(* Logix 5000 project; controller Drives_Line1 1756-L72 rev 20.13; software revision 20.04 *)

TASK Medium (periodic, rate 50 ms, priority 10, watchdog 1000 ms) : P00_Line, P01_Entry_Zone, P02_Exit_Zone, P10_Unwinder_1, P11_Unwinder_2, P12_Pinchroll_1, P13_Pinchroll_2, P14_Bridle_01

MODULES
   Local : 1756-L72 (ICP 0, rev 20.13)
      Master_Line_1 : 1756-L72 (ICP 5, rev 20.1, $099675bf$ RPI 20 ms, $797531a6$ RPI 20 ms, $6b587a51$ RPI 20 ms)
      EN2TR : vendor 1 type 12 code 200 (ICP 1, Ethernet 192.168.1.6, rev 3.1, Input RPI 500 ms)
         Drive_Bridle_04a : vendor 1 type 142 code 2192 (Ethernet 192.168.1.23, rev 7.1, Output RPI 20 ms)
             : vendor 1 type 142 code 8352 (RhinoBP 6, rev 1.6)
             : vendor 1 type 142 code 416 (RhinoBP 7, rev 1.8)
             : vendor 1 type 142 code 16544 (RhinoBP 5, rev 1.1)
             : vendor 1 type 142 code 24736 (RhinoBP 8, rev 1.1)
             : vendor 1 type 142 code 32928 (RhinoBP 13, rev 1.1)
             : vendor 1 type 142 code 33184 (RhinoBP 14, rev 2.5)
             : vendor 1 type 142 code 57760 (RhinoBP 4, rev 1.1)
         Drive_Pinchroll_2 : vendor 1 type 142 code 2192 (Ethernet 192.168.1.13, rev 7.1, Output RPI 20 ms)
             : vendor 1 type 142 code 416 (RhinoBP 7, rev 1.8)
             : vendor 1 type 142 code 57760 (RhinoBP 4, rev 1.1)
             : vendor 1 type 142 code 767 (RhinoBP 1, rev 2.2)
             : vendor 1 type 142 code 32928 (RhinoBP 13, rev 1.1)
             : vendor 1 type 142 code 24736 (RhinoBP 8, rev 1.1)
             : vendor 1 type 142 code 33184 (RhinoBP 14, rev 2.5)
             : vendor 1 type 142 code 8352 (RhinoBP 6, rev 1.6)
             : vendor 1 type 142 code 16544 (RhinoBP 5, rev 1.1)
         Drive_Pinchroll_3 : vendor 1 type 142 code 2192 (Ethernet 192.168.1.26, rev 5.1, Output RPI 20 ms)
             : vendor 1 type 142 code 33184 (RhinoBP 14, rev 2.4)
             : vendor 1 type 142 code 24736 (RhinoBP 8, rev 1.1)
             : vendor 1 type 142 code 16544 (RhinoBP 5, rev 1.1)
             : vendor 1 type 142 code 32928 (RhinoBP 13, rev 1.1)
             : vendor 1 type 142 code 8352 (RhinoBP 6, rev 1.6)
             : vendor 1 type 142 code 57760 (RhinoBP 4, rev 1.1)
             : vendor 1 type 142 code 416 (RhinoBP 7, rev 1.8)
         Drive_Bridle_02a : vendor 1 type 142 code 2192 (Ethernet 192.168.1.18, rev 7.1, Output RPI 20 ms)
             : vendor 1 type 142 code 416 (RhinoBP 7, rev 1.8)
             : vendor 1 type 142 code 16544 (RhinoBP 5, rev 1.1)
             : vendor 1 type 142 code 24736 (RhinoBP 8, rev 1.1)
             : vendor 1 type 142 code 33184 (RhinoBP 14, rev 2.5)
             : vendor 1 type 142 code 8352 (RhinoBP 6, rev 1.6)
             : vendor 1 type 142 code 32928 (RhinoBP 13, rev 1.1)
             : vendor 1 type 142 code 57760 (RhinoBP 4, rev 1.1)
         Drive_Unwinder_1 : vendor 1 type 142 code 2192 (Ethernet 192.168.1.10, rev 7.1, Output RPI 20 ms)
             : vendor 1 type 142 code 8352 (RhinoBP 6, rev 1.6)
             : vendor 1 type 142 code 33184 (RhinoBP 14, rev 2.5)
             : vendor 1 type 142 code 57760 (RhinoBP 4, rev 1.1)
             : vendor 1 type 142 code 32928 (RhinoBP 13, rev 1.1)
             : vendor 1 type 142 code 767 (RhinoBP 1, rev 2.2)
             : vendor 1 type 142 code 24736 (RhinoBP 8, rev 1.1)
             : vendor 1 type 142 code 416 (RhinoBP 7, rev 1.8)
             : vendor 1 type 142 code 16544 (RhinoBP 5, rev 1.1)
         Drive_Bridle_01a : vendor 1 type 142 code 2192 (Ethernet 192.168.1.14, rev 7.1, Output RPI 20 ms)
             : vendor 1 type 142 code 57760 (RhinoBP 4, rev 1.1)
             : vendor 1 type 142 code 16544 (RhinoBP 5, rev 1.1)
             : vendor 1 type 142 code 8352 (RhinoBP 6, rev 1.6)
             : vendor 1 type 142 code 33184 (RhinoBP 14, rev 2.5)
             : vendor 1 type 142 code 416 (RhinoBP 7, rev 1.8)
             : vendor 1 type 142 code 24736 (RhinoBP 8, rev 1.1)
             : vendor 1 type 142 code 32928 (RhinoBP 13, rev 1.1)
         Drive_Bridle_02b : vendor 1 type 142 code 2192 (Ethernet 192.168.1.19, rev 7.1, Output RPI 20 ms)
             : vendor 1 type 142 code 33184 (RhinoBP 14, rev 2.5)
             : vendor 1 type 142 code 24736 (RhinoBP 8, rev 1.1)
             : vendor 1 type 142 code 416 (RhinoBP 7, rev 1.8)
             : vendor 1 type 142 code 57760 (RhinoBP 4, rev 1.1)
             : vendor 1 type 142 code 16544 (RhinoBP 5, rev 1.1)
             : vendor 1 type 142 code 8352 (RhinoBP 6, rev 1.6)
             : vendor 1 type 142 code 32928 (RhinoBP 13, rev 1.1)
         Drive_Bridle_03a : vendor 1 type 142 code 2192 (Ethernet 192.168.1.20, rev 7.1, Output RPI 20 ms)
             : vendor 1 type 142 code 57760 (RhinoBP 4, rev 1.1)
             : vendor 1 type 142 code 8352 (RhinoBP 6, rev 1.6)
             : vendor 1 type 142 code 33184 (RhinoBP 14, rev 2.5)
             : vendor 1 type 142 code 32928 (RhinoBP 13, rev 1.1)
             : vendor 1 type 142 code 416 (RhinoBP 7, rev 1.8)
             : vendor 1 type 142 code 16544 (RhinoBP 5, rev 1.1)
             : vendor 1 type 142 code 24736 (RhinoBP 8, rev 1.1)
         Drive_Bridle_01c : vendor 1 type 142 code 2192 (Ethernet 192.168.1.16, rev 7.1, Output RPI 20 ms)
             : vendor 1 type 142 code 416 (RhinoBP 7, rev 1.8)
             : vendor 1 type 142 code 8352 (RhinoBP 6, rev 1.6)
             : vendor 1 type 142 code 32928 (RhinoBP 13, rev 1.1)
             : vendor 1 type 142 code 16544 (RhinoBP 5, rev 1.1)
             : vendor 1 type 142 code 24736 (RhinoBP 8, rev 1.1)
             : vendor 1 type 142 code 57760 (RhinoBP 4, rev 1.1)
             : vendor 1 type 142 code 33184 (RhinoBP 14, rev 2.5)
         Drive_Unwinder_2 : vendor 1 type 142 code 2192 (Ethernet 192.168.1.11, rev 7.1, Output RPI 20 ms)
             : vendor 1 type 142 code 416 (RhinoBP 7, rev 1.8)
             : vendor 1 type 142 code 24736 (RhinoBP 8, rev 1.1)
             : vendor 1 type 142 code 767 (RhinoBP 1, rev 2.2)
             : vendor 1 type 142 code 33184 (RhinoBP 14, rev 2.5)
             : vendor 1 type 142 code 57760 (RhinoBP 4, rev 1.1)
             : vendor 1 type 142 code 16544 (RhinoBP 5, rev 1.1)
             : vendor 1 type 142 code 8352 (RhinoBP 6, rev 1.6)
             : vendor 1 type 142 code 32928 (RhinoBP 13, rev 1.1)
         Drive_Bridle_01b : vendor 1 type 142 code 2192 (Ethernet 192.168.1.15, rev 7.1, Output RPI 20 ms)
             : vendor 1 type 142 code 57760 (RhinoBP 4, rev 1.1)
             : vendor 1 type 142 code 416 (RhinoBP 7, rev 1.8)
             : vendor 1 type 142 code 33184 (RhinoBP 14, rev 2.5)
             : vendor 1 type 142 code 8352 (RhinoBP 6, rev 1.6)
             : vendor 1 type 142 code 32928 (RhinoBP 13, rev 1.1)
             : vendor 1 type 142 code 16544 (RhinoBP 5, rev 1.1)
             : vendor 1 type 142 code 24736 (RhinoBP 8, rev 1.1)
         Drive_Pinchroll_1 : vendor 1 type 142 code 2192 (Ethernet 192.168.1.12, rev 7.1, Output RPI 20 ms)
             : vendor 1 type 142 code 57760 (RhinoBP 4, rev 1.1)
             : vendor 1 type 142 code 24736 (RhinoBP 8, rev 1.1)
             : vendor 1 type 142 code 16544 (RhinoBP 5, rev 1.1)
             : vendor 1 type 142 code 8352 (RhinoBP 6, rev 1.6)
             : vendor 1 type 142 code 33184 (RhinoBP 14, rev 2.5)
             : vendor 1 type 142 code 32928 (RhinoBP 13, rev 1.1)
             : vendor 1 type 142 code 416 (RhinoBP 7, rev 1.8)
         Drive_Bridle_03b : vendor 1 type 142 code 2192 (Ethernet 192.168.1.21, rev 7.1, Output RPI 20 ms)
             : vendor 1 type 142 code 32928 (RhinoBP 13, rev 1.1)
             : vendor 1 type 142 code 416 (RhinoBP 7, rev 1.8)
             : vendor 1 type 142 code 16544 (RhinoBP 5, rev 1.1)
             : vendor 1 type 142 code 57760 (RhinoBP 4, rev 1.1)
             : vendor 1 type 142 code 33184 (RhinoBP 14, rev 2.5)
             : vendor 1 type 142 code 8352 (RhinoBP 6, rev 1.6)
             : vendor 1 type 142 code 24736 (RhinoBP 8, rev 1.1)
         Drive_Winder : vendor 1 type 142 code 2192 (Ethernet 192.168.1.27, rev 7.1, Output RPI 20 ms)
             : vendor 1 type 142 code 24736 (RhinoBP 8, rev 1.1)
             : vendor 1 type 142 code 32928 (RhinoBP 13, rev 1.1)
             : vendor 1 type 142 code 416 (RhinoBP 7, rev 1.8)
             : vendor 1 type 142 code 8352 (RhinoBP 6, rev 1.6)
             : vendor 1 type 142 code 57760 (RhinoBP 4, rev 1.1)
             : vendor 1 type 142 code 33184 (RhinoBP 14, rev 2.5)
             : vendor 1 type 142 code 16544 (RhinoBP 5, rev 1.1)
         Drive_Bridle_04c : vendor 1 type 142 code 2192 (Ethernet 192.168.1.25, rev 7.1, Output RPI 20 ms)
             : vendor 1 type 142 code 57760 (RhinoBP 4, rev 1.1)
             : vendor 1 type 142 code 16544 (RhinoBP 5, rev 1.1)
             : vendor 1 type 142 code 33184 (RhinoBP 14, rev 2.5)
             : vendor 1 type 142 code 24736 (RhinoBP 8, rev 1.1)
             : vendor 1 type 142 code 416 (RhinoBP 7, rev 1.8)
             : vendor 1 type 142 code 8352 (RhinoBP 6, rev 1.6)
             : vendor 1 type 142 code 767 (RhinoBP 1, rev 2.2)
             : vendor 1 type 142 code 32928 (RhinoBP 13, rev 1.1)
         Drive_Entry_Accu : vendor 1 type 142 code 2192 (Ethernet 192.168.1.17, rev 9.1, Output RPI 20 ms)
             : vendor 1 type 142 code 57760 (RhinoBP 4, rev 1.1)
             : vendor 1 type 142 code 33184 (RhinoBP 14, rev 2.5)
             : vendor 1 type 142 code 24736 (RhinoBP 8, rev 1.1)
             : vendor 1 type 142 code 8352 (RhinoBP 6, rev 1.6)
             : vendor 1 type 142 code 16544 (RhinoBP 5, rev 1.1)
             : vendor 1 type 142 code 767 (RhinoBP 1, rev 2.2)
             : vendor 1 type 142 code 416 (RhinoBP 7, rev 1.8)
             : vendor 1 type 142 code 32928 (RhinoBP 13, rev 1.1)
         Drive_Exit_Accu : vendor 1 type 142 code 2192 (Ethernet 192.168.1.22, rev 7.1, Output RPI 20 ms)
             : vendor 1 type 142 code 33184 (RhinoBP 14, rev 2.5)
             : vendor 1 type 142 code 8352 (RhinoBP 6, rev 1.6)
             : vendor 1 type 142 code 416 (RhinoBP 7, rev 1.8)
             : vendor 1 type 142 code 24736 (RhinoBP 8, rev 1.1)
             : vendor 1 type 142 code 57760 (RhinoBP 4, rev 1.1)
             : vendor 1 type 142 code 16544 (RhinoBP 5, rev 1.1)
             : vendor 1 type 142 code 32928 (RhinoBP 13, rev 1.1)
         Drive_Bridle_04b : vendor 1 type 142 code 2192 (Ethernet 192.168.1.24, rev 7.1, Output RPI 20 ms)
             : vendor 1 type 142 code 416 (RhinoBP 7, rev 1.8)
             : vendor 1 type 142 code 16544 (RhinoBP 5, rev 1.1)
             : vendor 1 type 142 code 8352 (RhinoBP 6, rev 1.6)
             : vendor 1 type 142 code 57760 (RhinoBP 4, rev 1.1)
             : vendor 1 type 142 code 32928 (RhinoBP 13, rev 1.1)
             : vendor 1 type 142 code 33184 (RhinoBP 14, rev 2.5)
             : vendor 1 type 142 code 24736 (RhinoBP 8, rev 1.1)
         Drive_cu : PowerFlex 755-EENET (Ethernet 192.168.1.28, rev 9.1, Output RPI 20 ms)
             : vendor 1 type 143 code 767 (RhinoBP 1, rev 2.3)
             : vendor 1 type 143 code 9472 (RhinoBP 2, rev 1.4)
             : vendor 1 type 143 code 8352 (RhinoBP 6, rev 1.6)
             : vendor 1 type 143 code 32928 (RhinoBP 13, rev 1.1)
             : vendor 1 type 143 code 33184 (RhinoBP 14, rev 2.5)
             : vendor 1 type 143 code 416 (RhinoBP 4, rev 1.8)
             : vendor 1 type 143 code 16544 (RhinoBP 5, rev 1.1)
END_MODULES

TYPE UDT_Bridle_2M :
STRUCT
   PF755_shaft_a : UDT_PF755;
   PF755_shaft_b : UDT_PF755;
   Cmd : UDT_Commands_Bridle;
   Stat : UDT_Status_Bridle;
   Ctrl : UDT_Control_Bridle_2M;
   Fbdk_shaft_a : UDT_Feedbacks_Bridle;
   Fbdk_shaft_b : UDT_Feedbacks_Bridle;
   Config_shaft_a : UDT_Config_Bridle;
   Config_shaft_b : UDT_Config_Bridle;
   SpdTrim_MPS : REAL;
   SpdTrim_Pct : REAL;
END_STRUCT
END_TYPE

TYPE UDT_Bridle_3M :
STRUCT
   PF755_shaft_a : UDT_PF755;
   PF755_shaft_b : UDT_PF755;
   PF755_shaft_c : UDT_PF755;
   Stat : UDT_Status_Bridle;
   Fbdk_shaft_a : UDT_Feedbacks_Bridle;
   Fbdk_shaft_b : UDT_Feedbacks_Bridle;
   Fbdk_shaft_c : UDT_Feedbacks_Bridle;
   Config_shaft_a : UDT_Config_Bridle;
   Config_shaft_b : UDT_Config_Bridle;
   Config_shaft_c : UDT_Config_Bridle;
END_STRUCT
END_TYPE

TYPE UDT_Commands :
STRUCT
   Line : UDT_Commands_Line;
   Entry : UDT_Commands_Zone;
   Exit : UDT_Commands_Zone;
   Unwinder_1 : UDT_Commands_Unwinder;
   Unwinder_2 : UDT_Commands_Unwinder;
   Pinchroll_1 : UDT_Commands_Pinch;
   Pinchroll_2 : UDT_Commands_Pinch;
   Entry_Accu : UDT_Commands_Accu;
   Bridle_02 : UDT_Commands_Bridle;
   Bridle_03 : UDT_Commands_Bridle;
   Exit_Accu : UDT_Commands_Accu;
   PinchRoll_3 : UDT_Commands_Pinch;
   Winder : UDT_Commands_Winder;
   cu : UDT_Commands_Pinch;
END_STRUCT
END_TYPE

TYPE UDT_Commands_Accu :
STRUCT
   Run : BOOL;
   JogFwd : BOOL;
   JogRev : BOOL;
END_STRUCT
END_TYPE

TYPE UDT_Commands_Bridle :
STRUCT
   Run : BOOL;
   JogFwd : BOOL;
   JogRev : BOOL;
END_STRUCT
END_TYPE

TYPE UDT_Commands_Line :
STRUCT
   Run : BOOL;
   JogFwd : BOOL;
   JogRev : BOOL;
   ResetDrv : BOOL;
   WD_FromMaster : BOOL;
   ApplyFastStop : BOOL;
END_STRUCT
END_TYPE

TYPE UDT_Commands_Pinch :
STRUCT
   Run : BOOL;
   Coupled_shaft_1 : BOOL;
   Coupled_shaft_2 : BOOL;
   JogFwd : BOOL;
   JogRev : BOOL;
   MtrCb : BOOL;
END_STRUCT
END_TYPE

TYPE UDT_Commands_Unwinder :
STRUCT
   RunFwd : BOOL;
   RunRev : BOOL;
   JogFwd : BOOL;
   JogRev : BOOL;
   SetNewDiameter : BOOL;
   HeadToStitch : BOOL;
   HeadToShear : BOOL;
   ResetCoilLength : BOOL;
END_STRUCT
END_TYPE

TYPE UDT_Commands_Winder :
STRUCT
   RunFwd : BOOL;
   RunRev : BOOL;
   JogFwd : BOOL;
   JogRev : BOOL;
   SetNewDiameter : BOOL;
   ResetCoilLength : BOOL;
END_STRUCT
END_TYPE

TYPE UDT_Commands_Zone :
STRUCT
   Run : BOOL;
   JogFwd : BOOL;
   JogRev : BOOL;
   EndToShear : BOOL;
   EndToStitch : BOOL;
   HeadToStitch : BOOL;
   EndToCoiler : BOOL;
   NewStitch : BOOL;
END_STRUCT
END_TYPE

TYPE UDT_Config :
STRUCT
   Unwinder_1 : UDT_Config_Unwinder;
   Unwinder_2 : UDT_Config_Unwinder;
   Pinchroll_1 : UDT_Config_Pinch;
   Pinchroll_2 : UDT_Config_Pinch;
   Entry_Accu : UDT_Config_Accu;
   Bridle_01a : UDT_Config_Bridle;
   Bridle_01b : UDT_Config_Bridle;
   Bridle_01c : UDT_Config_Bridle;
   Bridle_02a : UDT_Config_Bridle;
   Bridle_02b : UDT_Config_Bridle;
   Bridle_03a : UDT_Config_Bridle;
   Bridle_03b : UDT_Config_Bridle;
   Bridle_04a : UDT_Config_Bridle;
   Bridle_04b : UDT_Config_Bridle;
   Bridle_04c : UDT_Config_Bridle;
   Exit_Accu : UDT_Config_Accu;
   PinchRoll_3 : UDT_Config_Pinch;
   Winder : UDT_Config_Winder;
   Entry : UDT_Config_Zone;
   Exit : UDT_Config_Zone;
   Line : UDT_Config_Line;
END_STRUCT
END_TYPE

TYPE UDT_Config_Accu :
STRUCT
   zGearRatio : REAL;
   zMaxPos : REAL;
   zMinPos : REAL;
   zSyncPos : REAL;
   zJogRef : REAL;
   zAccJog : REAL;
   zDecJog : REAL;
   zJerkJog : REAL;
END_STRUCT
END_TYPE

TYPE UDT_Config_Bridle :
STRUCT
   zGearRatio : REAL;
   DiameterRoll : REAL;
END_STRUCT
END_TYPE

TYPE UDT_Config_Line :
STRUCT
   zAccRate : REAL;
   zDecRate : REAL;
   zJerk : REAL;
   zJogSpd : REAL;
   zJogAccRate : REAL;
   zJogDecRate : REAL;
   zMaxAccDec : REAL;
   zSpdMax : REAL;
END_STRUCT
END_TYPE

TYPE UDT_Config_Pinch :
STRUCT
   zGearRatio : REAL;
   DiameterRoll : REAL;
   zMaxAcc : REAL;
   zMaxDec : REAL;
   zJogRef : REAL;
   zAccJog : REAL;
   zDecJog : REAL;
   zJerkJog : REAL;
END_STRUCT
END_TYPE

TYPE UDT_Config_TM :
STRUCT
   zMinTen : REAL;
   zMaxTen : REAL;
END_STRUCT
END_TYPE

TYPE UDT_Config_Unwinder :
STRUCT
   zGearRatio : REAL;
   zMinDiameter : REAL;
   zMaxDiameter : REAL;
   zMinTension : REAL;
   zMaxTension : REAL;
   zJogRef : REAL;
   zDiamCalcEnblThresh_MPS : REAL;
   zDiamCalcUpdate_Rev : REAL;
   zMotorPwr : REAL;
   zMtrBaseSpd : REAL;
   zAccJog : REAL;
   zDecJog : REAL;
   zJerkJog : REAL;
END_STRUCT
END_TYPE

TYPE UDT_Config_Winder :
STRUCT
   zGearRatio : REAL;
   zMinDiameter : REAL;
   zMaxDiameter : REAL;
   zMinTension : REAL;
   zMaxTension : REAL;
   zJogRef : REAL;
   zDiamCalcEnblThresh_MPS : REAL;
   zDiamCalcUpdate_Rev : REAL;
   zMotorPwr : REAL;
   zMtrBaseSpd : REAL;
   zAccJog : REAL;
   zDecJog : REAL;
   zJerkJog : REAL;
END_STRUCT
END_TYPE

TYPE UDT_Config_Zone :
STRUCT
   zJogRef : REAL;
   zAccJog : REAL;
   zDecJog : REAL;
   zJerkJog : REAL;
   zAccRun : REAL;
   zDecRun : REAL;
   zJerkRun : REAL;
   zMaxAccDec : REAL;
   zMaxSpd : REAL;
END_STRUCT
END_TYPE

TYPE UDT_Control_Accu :
STRUCT
   Run : BOOL;
   JogFwd : BOOL;
   JogRev : BOOL;
   RmpdRefEnable : BOOL;
   URmpdRefEnable : BOOL;
   StartRamp : BOOL;
   TenRegOn : BOOL;
   PosRegOn : BOOL;
   SetSyncPos : BOOL;
   PosRegOutSpd : REAL;
   SpdTrim : REAL;
   FB_CountsPerMM : DINT;
END_STRUCT
END_TYPE

TYPE UDT_Control_Bridle_2M :
STRUCT
   JogFwd : BOOL;
   JogRev : BOOL;
   StartRamp : BOOL;
   RmpdRefEnable : BOOL;
   URmpdRefEnable : BOOL;
   zJogSpd : REAL;
   zJogAccRate : REAL;
   zJogDecRate : REAL;
   zJogJerkRate : REAL;
   zMaxAccDec : REAL;
END_STRUCT
END_TYPE

TYPE UDT_Control_Line :
STRUCT
   Run : BOOL;
   JogFwd : BOOL;
   JogRev : BOOL;
   StartRamp : BOOL;
   RmpdRefEnable : BOOL;
   URmpdRefEnable : BOOL;
   ApplyFastStop : BOOL;
   TenRegOn : BOOL;
   SpdRefRmp : REAL;
END_STRUCT
END_TYPE

TYPE UDT_Control_Pinch :
STRUCT
   Run : BOOL;
   Coupled_shaft_1 : BOOL;
   Coupled_shaft_2 : BOOL;
   JogFwd : BOOL;
   JogRev : BOOL;
   RmpdRefEnable : BOOL;
   URmpdRefEnable : BOOL;
   StartRamp : BOOL;
END_STRUCT
END_TYPE

TYPE UDT_Control_Unwind :
STRUCT
   JogFwd : BOOL;
   JogRev : BOOL;
   RunFwd : BOOL;
   RunRev : BOOL;
   TenRefStallEnbl : BOOL;
   TrimOn : BOOL;
   TrimPos : BOOL;
   TrimNeg : BOOL;
   TenRefOn : BOOL;
   DiamCalcIncEnbl : BOOL;
   DiamCalcDecEnbl : BOOL;
   TensionRef : REAL;
   RunSpdRef : REAL;
   RunSpdRefRate : REAL;
   RunSpdTrim : REAL;
   StartRamp : BOOL;
   RmpdRefEnable : BOOL;
   URmpdRefEnable : BOOL;
   BR : BOOL;
   Fan : BOOL;
END_STRUCT
END_TYPE

TYPE UDT_Control_Winder :
STRUCT
   JogFwd : BOOL;
   JogRev : BOOL;
   RunFwd : BOOL;
   RunRev : BOOL;
   TenRefStallEnbl : BOOL;
   TrimPos : BOOL;
   TrimNeg : BOOL;
   TrimOn : BOOL;
   TenRefOn : BOOL;
   DiamCalcIncEnbl : BOOL;
   DiamCalcDecEnbl : BOOL;
   TensionRef : REAL;
   RunSpdRef : REAL;
   RunSpdRefRate : REAL;
   RunSpdTrim : REAL;
   StartRamp : BOOL;
   RmpdRefEnable : BOOL;
   URmpdRefEnable : BOOL;
   BR : BOOL;
   Fan : BOOL;
END_STRUCT
END_TYPE

TYPE UDT_Control_Zone :
STRUCT
   Run : BOOL;
   JogFwd : BOOL;
   JogRev : BOOL;
   EndToShear : BOOL;
   EndToStitch : BOOL;
   EndToCoiler : BOOL;
   HeadToStitch : BOOL;
   StartRamp : BOOL;
   RmpdRefEnable : BOOL;
   URmpdRefEnable : BOOL;
   ApplyFastStop : BOOL;
   EOC_PosRedef : DINT;
   HOC_PosRedef : DINT;
   SpdRefRmp : REAL;
END_STRUCT
END_TYPE

TYPE UDT_Datalinks_in :
STRUCT
   OutputFrequency : REAL;
   OutputCurrent : REAL;
   OutputVoltage : REAL;
   OutputPower : REAL;
   SRegOutput : REAL;
   PTP_Feedback : DINT;
   LimitedTrqRef : REAL;
   FaultStatusA : DINT;
   FaultStatusB : DINT;
   StartInhibits : DINT;
   P7_Ptc_Sts : DINT;
   P7_DigitalOutSts : DINT;
   P7_DigitalInSts : DINT;
   HomingStatus : DINT;
END_STRUCT
END_TYPE

TYPE UDT_Datalinks_Out :
STRUCT
   TorqueStep : REAL;
   TorqueSp : REAL;
   RegulatorMode : DINT;
   SpeedRegBW : REAL;
   HomingControl : DINT;
   UserHomePos : DINT;
   PID_Setpoint : REAL;
   SpdRegNegLim : REAL;
   SpdRegPosLim : REAL;
   PID_Ctrl : DINT;
   P7_DigOutSetpoint : DINT;
END_STRUCT
END_TYPE

TYPE UDT_Drive_Commands :
STRUCT
   LogicCommand : DINT;
   Stop : BOOL;
   Start : BOOL;
   Jog1 : BOOL;
   ClearFaults : BOOL;
   Forward : BOOL;
   Reverse : BOOL;
   Manual : BOOL;
   AccelTime1 : BOOL;
   AccelTime2 : BOOL;
   DecelTime1 : BOOL;
   DecelTime2 : BOOL;
   SpdRefSel0 : BOOL;
   SpdRefSel1 : BOOL;
   SpdRefSel2 : BOOL;
   CoastStop : BOOL;
   CLimitStop : BOOL;
   Run : BOOL;
   Jog2 : BOOL;
   Reference : REAL;
END_STRUCT
END_TYPE

TYPE UDT_Drive_Status :
STRUCT
   Drive_status : DINT;
   Ready : BOOL;
   Active : BOOL;
   CommandDir : BOOL;
   ActualDir : BOOL;
   Accelerating : BOOL;
   Decelerating : BOOL;
   Alarm : BOOL;
   Faulted : BOOL;
   AtSpeed : BOOL;
   Manual : BOOL;
   SpdRefBit0 : BOOL;
   SpdRefBit1 : BOOL;
   SpdRefBit2 : BOOL;
   SpdRefBit3 : BOOL;
   SpdRefBit4 : BOOL;
   Running : BOOL;
   Jogging : BOOL;
   Stopping : BOOL;
   DCBraking : BOOL;
   DBActive : BOOL;
   SpeedMode : BOOL;
   PositionMode : BOOL;
   TorqueMode : BOOL;
   AtZeroSpeed : BOOL;
   AtHome : BOOL;
   AtLimit : BOOL;
   CurrLimit : BOOL;
   BusFrqReg : BOOL;
   EnableOn : BOOL;
   MotorOL : BOOL;
   Regen : BOOL;
   Feedback : REAL;
END_STRUCT
END_TYPE

TYPE UDT_Entry_Accu :
STRUCT
   PF755 : UDT_PF755;
   Cmd : UDT_Commands_Accu;
   Stat : UDT_Status_Accu;
   Fdbk : UDT_Feedbacks_Accu;
   Sp : UDT_Setpoints_Accu;
   Config : UDT_Config_Accu;
   Ctrl : UDT_Control_Accu;
END_STRUCT
END_TYPE

TYPE UDT_Exit_Accu :
STRUCT
   PF755 : UDT_PF755;
   Cmd : UDT_Commands_Accu;
   Stat : UDT_Status_Accu;
   Fdbk : UDT_Feedbacks_Accu;
   Sp : UDT_Setpoints_Accu;
   Config : UDT_Config_Accu;
   Ctrl : UDT_Control_Accu;
END_STRUCT
END_TYPE

TYPE UDT_Fdbks :
STRUCT
   Unwinder_1 : UDT_Feedbacks_Unwinder;
   Unwinder_2 : UDT_Feedbacks_Unwinder;
   Pinchroll_1 : UDT_Feedbacks_Pinch;
   Pinchroll_2 : UDT_Feedbacks_Pinch;
   Entry_Accu : UDT_Feedbacks_Accu;
   Bridle_01a : UDT_Feedbacks_Bridle;
   Bridle_01b : UDT_Feedbacks_Bridle;
   Bridle_01c : UDT_Feedbacks_Bridle;
   Bridle_02a : UDT_Feedbacks_Bridle;
   Bridle_02b : UDT_Feedbacks_Bridle;
   Bridle_03a : UDT_Feedbacks_Bridle;
   Bridle_03b : UDT_Feedbacks_Bridle;
   Bridle_04a : UDT_Feedbacks_Bridle;
   Bridle_04b : UDT_Feedbacks_Bridle;
   Bridle_04c : UDT_Feedbacks_Bridle;
   Exit_Accu : UDT_Feedbacks_Accu;
   Pinchroll_3 : UDT_Feedbacks_Pinch;
   Winder : UDT_Feedbacks_Winder;
   Line : UDT_Feedbacks_Line;
   Entry : UDT_Feedbacks_Zone;
   Exit : UDT_Feedbacks_Zone;
   cu : UDT_Feedbacks_Pinch;
END_STRUCT
END_TYPE

TYPE UDT_Feedbacks_Accu :
STRUCT
   PvSpeed : REAL;
   PvActualPos : REAL;
   PvActualPosPct : REAL;
   PvSpdRef_MPS : REAL;
   PvSpdRef_RPM : REAL;
END_STRUCT
END_TYPE

TYPE UDT_Feedbacks_Bridle :
STRUCT
   PvSurfaceSpeed : REAL;
   SpSpdRef_MPS : REAL;
END_STRUCT
END_TYPE

TYPE UDT_Feedbacks_Line :
STRUCT
   LineSpeed : REAL;
   Stitch_Cntrs : UDT_Stitch_Counter;
END_STRUCT
END_TYPE

TYPE UDT_Feedbacks_Pinch :
STRUCT
   PvSurfaceSpeed : REAL;
   PvSpdRef_MPS : REAL;
   PvSpdRef_RPM : REAL;
END_STRUCT
END_TYPE

TYPE UDT_Feedbacks_Unwinder :
STRUCT
   PvSurfaceSpeed : REAL;
   PvActualDiameter : REAL;
   PvTension : REAL;
   PvSpdRef_MPS : REAL;
   PvNormInertia : REAL;
   PvTotalInertia : REAL;
   PvRpm : REAL;
   PvSpdRef_RPM : REAL;
   PvTrimSpdRef : REAL;
   PvCoilLength : REAL;
END_STRUCT
END_TYPE

TYPE UDT_Feedbacks_Winder :
STRUCT
   PvSurfaceSpeed : REAL;
   PvActualDiameter : REAL;
   PvTension : REAL;
   PvSpdRef_MPS : REAL;
   PvNormInertia : REAL;
   PvTotalInertia : REAL;
   PvRpm : REAL;
   PvSpdRef_RPM : REAL;
   PvTrimSpdRef : REAL;
   PvCoilLength : REAL;
END_STRUCT
END_TYPE

TYPE UDT_Feedbacks_Zone :
STRUCT
   PvActualSpeed : REAL;
   PvSpeedRef : REAL;
END_STRUCT
END_TYPE

TYPE UDT_PF755 :
STRUCT
   DL_In : UDT_Datalinks_in;
   DL_Out : UDT_Datalinks_Out;
   IO_ConnectionOk : BOOL;
   NoResponse : BOOL;
   Feedback : REAL;
   Reference : REAL;
END_STRUCT
END_TYPE

TYPE UDT_Pinchroll :
STRUCT
   PF755 : UDT_PF755;
   Cmd : UDT_Commands_Pinch;
   Stat : UDT_Status_Pinch;
   Fdbk : UDT_Feedbacks_Pinch;
   Config : UDT_Config_Pinch;
   Ctrl : UDT_Control_Pinch;
END_STRUCT
END_TYPE

TYPE UDT_Setpoints :
STRUCT
   Unwinder_1 : UDT_Setpoints_Unwinder;
   Unwinder_2 : UDT_Setpoints_Unwinder;
   Entry_Accu : UDT_Setpoints_Accu;
   Exit_Accu : UDT_Setpoints_Accu;
   Winder : UDT_Setpoints_Winder;
   TM1 : UDT_Setpoints_TM;
   TM2 : UDT_Setpoints_TM;
   TM3 : UDT_Setpoints_TM;
   Line : UDT_Setpoints_Line;
   Entry : UDT_Setpoints_Zone;
   Exit : UDT_Setpoints_Zone;
END_STRUCT
END_TYPE

TYPE UDT_Setpoints_Accu :
STRUCT
   SpPos : REAL;
END_STRUCT
END_TYPE

TYPE UDT_Setpoints_Line :
STRUCT
   RunSpdRef : REAL;
   WebWidth : REAL;
   MaterialDensity : REAL;
   SpMmPerRev : REAL;
   JogSpdRef : REAL;
END_STRUCT
END_TYPE

TYPE UDT_Setpoints_TM :
STRUCT
   SpTen : REAL;
   PvTen : REAL;
   MaxTen : REAL;
   MinTen : REAL;
END_STRUCT
END_TYPE

TYPE UDT_Setpoints_Unwinder :
STRUCT
   SpNewDiameter : REAL;
   SpTension : REAL;
   zCellToStitch : REAL;
   zCellToShear : REAL;
END_STRUCT
END_TYPE

TYPE UDT_Setpoints_Winder :
STRUCT
   SpNewDiameter : REAL;
   SpTension : REAL;
   zCellToStitch : REAL;
   zCellToShear : REAL;
END_STRUCT
END_TYPE

TYPE UDT_Setpoints_Zone :
STRUCT
   MaxSpdRef : REAL;
END_STRUCT
END_TYPE

TYPE UDT_Status :
STRUCT
   Line : UDT_Status_Line;
   Entry : UDT_Status_Zone;
   Exit : UDT_Status_Zone;
   Unwinder_1 : UDT_Status_Unwinder;
   Unwinder_2 : UDT_Status_Unwinder;
   Pinchroll_1 : UDT_Status_Pinch;
   Pinchroll_2 : UDT_Status_Pinch;
   Entry_Accu : UDT_Status_Accu;
   Bridle_01 : UDT_Status_Bridle;
   Bridle_02 : UDT_Status_Bridle;
   Bridle_03 : UDT_Status_Bridle;
   Bridle_04 : UDT_Status_Bridle;
   Exit_Accu : UDT_Status_Accu;
   Pinchroll_3 : UDT_Status_Pinch;
   Winder : UDT_Status_Winder;
   TM1 : UDT_Status_TM;
   TM2 : UDT_Status_TM;
   TM3 : UDT_Status_TM;
   cu : UDT_Status_Pinch;
END_STRUCT
END_TYPE

TYPE UDT_Status_Accu :
STRUCT
   RunningFwd : BOOL;
   RunningRev : BOOL;
   JoggingFwd : BOOL;
   JoggingRev : BOOL;
   Running : BOOL;
   Stopped : BOOL;
   Held : BOOL;
   BrOk : BOOL;
   CB_Ok : BOOL;
   SafetyOk : BOOL;
   NoFastStop : BOOL;
   NoPrecharge : BOOL;
   Ready : BOOL;
   NoOverTemp : BOOL;
   FanOn : BOOL;
   BrakeOff : BOOL;
   Synch : BOOL;
   TenRegOnSp : BOOL;
   Full : BOOL;
   Empty : BOOL;
   NotAtLimit : BOOL;
   LowTension : BOOL;
END_STRUCT
END_TYPE

TYPE UDT_Status_Bridle :
STRUCT
   RunningFwd : BOOL;
   RunningRev : BOOL;
   JoggingFwd : BOOL;
   JoggingRev : BOOL;
   Stopped : BOOL;
   Held : BOOL;
   Running : BOOL;
   Faulted : BOOL;
   AllActive : BOOL;
   AllEnabled : BOOL;
   AllStopped : BOOL;
   AllHolded : BOOL;
   AllSelected : BOOL;
   AllStandStill : BOOL;
   All_CB_Ok : BOOL;
   All_BrakeResOk : BOOL;
   AllSafetyOk : BOOL;
   NoFastStop : BOOL;
   NoPrecharge : BOOL;
   AllReady : BOOL;
   NoOverTemp : BOOL;
   AllFanOn : BOOL;
   AllBrakeOff : BOOL;
   IOConnOkAllDrvs : BOOL;
   FanOn : BOOL;
   BrakeOff : BOOL;
   TenRegOnSp : BOOL;
   LowTension : BOOL;
END_STRUCT
END_TYPE

TYPE UDT_Status_Line :
STRUCT
   AllDrivesEnabled : BOOL;
   AllDrivesActive : BOOL;
   SafetyOkAllDrvs : BOOL;
   AllDrivesAtZeroSpd : BOOL;
   WD_ToMaster : BOOL;
   Entry_drives_ready : BOOL;
   Exit_drives_ready : BOOL;
   MasterPlcOk : BOOL;
   DrivesReady : BOOL;
   LineReady : BOOL;
   NoFastStop : BOOL;
   TensionOk : BOOL;
   Running : BOOL;
   JoggingFwd : BOOL;
   JoggingRev : BOOL;
   ApplyFastStop : BOOL;
   AllStandstill : BOOL;
END_STRUCT
END_TYPE

TYPE UDT_Status_Pinch :
STRUCT
   Coupled_shaft_1 : BOOL;
   Coupled_shaft_2 : BOOL;
   RunningFwd : BOOL;
   RunningRev : BOOL;
   Running : BOOL;
   JoggingFwd : BOOL;
   JoggingRev : BOOL;
   Selected : BOOL;
   Stopped : BOOL;
   Held : BOOL;
   CB_Ok : BOOL;
   SafetyOk : BOOL;
   NoFastStop : BOOL;
   NoPrecharge : BOOL;
   Ready : BOOL;
   NoOverTemp : BOOL;
   FanOn : BOOL;
   BrakeOff : BOOL;
   Sync : BOOL;
END_STRUCT
END_TYPE

TYPE UDT_Status_TM :
STRUCT
   RegOnSp : BOOL;
   RegOutOfLim : BOOL;
END_STRUCT
END_TYPE

TYPE UDT_Status_Unwinder :
STRUCT
   RunningFwd : BOOL;
   RunningRev : BOOL;
   JoggingFwd : BOOL;
   JoggingRev : BOOL;
   Running : BOOL;
   Stopped : BOOL;
   Selected : BOOL;
   Held : BOOL;
   NewDiameterActive : BOOL;
   CB_Ok : BOOL;
   SafetyOk : BOOL;
   NoFastStop : BOOL;
   NoPrecharge : BOOL;
   Ready : BOOL;
   NoOverTemp : BOOL;
   FanOn : BOOL;
   BrakeOff : BOOL;
   DiameterCalcEnbl : BOOL;
   TensRegOnSp : BOOL;
   LowTension : BOOL;
   HeadAtStitch : BOOL;
   RollEmpty : BOOL;
END_STRUCT
END_TYPE

TYPE UDT_Status_Winder :
STRUCT
   RunningFwd : BOOL;
   RunningRev : BOOL;
   JoggingFwd : BOOL;
   JoggingRev : BOOL;
   Running : BOOL;
   Stopped : BOOL;
   Selected : BOOL;
   Held : BOOL;
   NewDiameterActive : BOOL;
   CB_Ok : BOOL;
   SafetyOk : BOOL;
   NoFastStop : BOOL;
   NoPrecharge : BOOL;
   Ready : BOOL;
   NoOverTemp : BOOL;
   FanOn : BOOL;
   BrakeOff : BOOL;
   DiameterCalcEnbl : BOOL;
   TensRegOnSp : BOOL;
   LowTension : BOOL;
   EndAtStitch : BOOL;
   EndAtShear : BOOL;
   RollFull : BOOL;
END_STRUCT
END_TYPE

TYPE UDT_Status_Zone :
STRUCT
   AllDrivesEnabled : BOOL;
   IOConnOkDrives : BOOL;
   NoFastStop : BOOL;
   AllDrivesActive : BOOL;
   SafetyOkAllDrvs : BOOL;
   AllDrivesAtZeroSpd : BOOL;
   DrivesReady : BOOL;
   TensionOk : BOOL;
   Running : BOOL;
   RunningFwd : BOOL;
   RunningRev : BOOL;
   JoggingFwd : BOOL;
   JoggingRev : BOOL;
   Standstilll : BOOL;
   BR_Ok : BOOL;
   All_CB_Ok : BOOL;
   Ready : BOOL;
   EndAtStitch : BOOL;
   EndAtShear : BOOL;
   HeadAtStitch : BOOL;
   HeadAtShear : BOOL;
   EndAtCoiler : BOOL;
END_STRUCT
END_TYPE

TYPE UDT_Stitch_Counter :
STRUCT
   Zone_1 : REAL[3];
   Zone_2 : REAL[5];
   Zone_3 : REAL;
END_STRUCT
END_TYPE

TYPE UDT_TM :
STRUCT
   Sp : UDT_Setpoints_TM;
   Stat : UDT_Status_TM;
END_STRUCT
END_TYPE

TYPE UDT_Unwinder :
STRUCT
   PF755 : UDT_PF755;
   Cmd : UDT_Commands_Unwinder;
   Stat : UDT_Status_Unwinder;
   Fdbk : UDT_Feedbacks_Unwinder;
   Sp : UDT_Setpoints_Unwinder;
   Config : UDT_Config_Unwinder;
   Ctrl : UDT_Control_Unwind;
END_STRUCT
END_TYPE

TYPE UDT_Winder :
STRUCT
   PF755 : UDT_PF755;
   Cmd : UDT_Commands_Winder;
   Stat : UDT_Status_Winder;
   Fdbk : UDT_Feedbacks_Winder;
   Sp : UDT_Setpoints_Winder;
   Config : UDT_Config_Winder;
   Ctrl : UDT_Control_Winder;
END_STRUCT
END_TYPE

VAR_GLOBAL   (* controller tags *)
   _bob : BOOL;
   _bv_tmp : INT := 1030;
   Bridle_01 : UDT_Bridle_3M := (PF755_shaft_a.DL_In.PTP_Feedback := 19942566, PF755_shaft_a.DL_In.P7_Ptc_Sts := 1, PF755_shaft_a.DL_In.P7_DigitalInSts := 2#0000_0000_0000_0000_0000_0000_0000_0111, PF755_shaft_a.IO_ConnectionOk := 1, PF755_shaft_b.DL_In.PTP_Feedback := 9220666, PF755_shaft_b.DL_In.P7_Ptc_Sts := 1, PF755_shaft_b.DL_In.P7_DigitalInSts := 2#0000_0000_0000_0000_0000_0000_0000_0111, PF755_shaft_b.IO_ConnectionOk := 1, PF755_shaft_c.DL_In.PTP_Feedback := 531146554, PF755_shaft_c.DL_In.P7_Ptc_Sts := 4, PF755_shaft_c.DL_In.P7_DigitalInSts := 2#0000_0000_0000_0000_0000_0000_0000_0011, PF755_shaft_c.IO_ConnectionOk := 1, Stat.Stopped := 1, Stat.AllEnabled := 1, Stat.AllStandStill := 1, Stat.All_CB_Ok := 1, Stat.AllSafetyOk := 1, Stat.NoFastStop := 1, Stat.NoPrecharge := 1, Stat.AllReady := 1, Stat.NoOverTemp := 1, Stat.IOConnOkAllDrvs := 1, Config_shaft_a.zGearRatio := 129.41, Config_shaft_a.DiameterRoll := 801.0, Config_shaft_b.zGearRatio := 129.41, Config_shaft_b.DiameterRoll := 801.0, Config_shaft_c.zGearRatio := 27.88, Config_shaft_c.DiameterRoll := 202.12);
   Bridle_01_FB_Diff : REAL;
   Bridle_01_FB_Update_Valid : BOOL;
   Bridle_01_Rev_mm : REAL := 0.05142632;
   Bridle_01b_FBCounts_mm : REAL := 210.64221;
   Bridle_02 : UDT_Bridle_2M := (PF755_shaft_a.DL_In.PTP_Feedback := -464433170, PF755_shaft_a.DL_In.P7_Ptc_Sts := 1, PF755_shaft_a.DL_In.P7_DigitalInSts := 2#0000_0000_0000_0000_0000_0000_0000_0011, PF755_shaft_a.IO_ConnectionOk := 1, PF755_shaft_a.Reference := 4.284751, PF755_shaft_b.DL_In.PTP_Feedback := -486222257, PF755_shaft_b.DL_In.P7_Ptc_Sts := 1, PF755_shaft_b.DL_In.P7_DigitalInSts := 2#0000_0000_0000_0000_0000_0000_0000_0011, PF755_shaft_b.IO_ConnectionOk := 1, PF755_shaft_b.Reference := 4.284751, Stat.Stopped := 1, Stat.AllEnabled := 1, Stat.AllStandStill := 1, Stat.All_CB_Ok := 1, Stat.AllSafetyOk := 1, Stat.NoFastStop := 1, Stat.NoPrecharge := 1, Stat.AllReady := 1, Stat.NoOverTemp := 1, Stat.IOConnOkAllDrvs := 1, Ctrl.zJogSpd := 0.083, Ctrl.zJogAccRate := 0.083, Ctrl.zJogDecRate := 0.083, Ctrl.zJogJerkRate := 0.1, Ctrl.zMaxAccDec := 0.25, Fbdk_shaft_a.SpSpdRef_MPS := 0.00068994303, Fbdk_shaft_b.SpSpdRef_MPS := 0.00068994303, Config_shaft_a.zGearRatio := 260.52, Config_shaft_a.DiameterRoll := 801.18, Config_shaft_b.zGearRatio := 260.52, Config_shaft_b.DiameterRoll := 801.18);
   Bridle_02_FB_Diff : DINT;
   Bridle_02_FB_Update_Valid : BOOL;
   Bridle_02_Rev_mm : REAL := 0.10350494;
   Bridle_02b_FBCounts_mm : DINT := 424;
   Bridle_03 : UDT_Bridle_2M := (PF755_shaft_a.DL_In.PTP_Feedback := -468415885, PF755_shaft_a.DL_In.P7_Ptc_Sts := 1, PF755_shaft_a.DL_In.P7_DigitalInSts := 2#0000_0000_0000_0000_0000_0000_0000_0011, PF755_shaft_a.IO_ConnectionOk := 1, PF755_shaft_a.Reference := 4.217773, PF755_shaft_b.DL_In.PTP_Feedback := -456701981, PF755_shaft_b.DL_In.P7_Ptc_Sts := 1, PF755_shaft_b.DL_In.P7_DigitalInSts := 2#0000_0000_0000_0000_0000_0000_0000_0011, PF755_shaft_b.IO_ConnectionOk := 1, PF755_shaft_b.Reference := 4.217773, Stat.Stopped := 1, Stat.AllEnabled := 1, Stat.AllStandStill := 1, Stat.All_CB_Ok := 1, Stat.AllSafetyOk := 1, Stat.NoFastStop := 1, Stat.NoPrecharge := 1, Stat.AllReady := 1, Stat.NoOverTemp := 1, Stat.IOConnOkAllDrvs := 1, Ctrl.zJogSpd := 0.083, Ctrl.zJogAccRate := 0.083, Ctrl.zJogDecRate := 0.083, Ctrl.zJogJerkRate := 0.1, Ctrl.zMaxAccDec := 0.25, Fbdk_shaft_a.SpSpdRef_MPS := 0.00068994303, Fbdk_shaft_b.SpSpdRef_MPS := 0.00068994303, Config_shaft_a.zGearRatio := 256.39, Config_shaft_a.DiameterRoll := 801.0, Config_shaft_b.zGearRatio := 256.39, Config_shaft_b.DiameterRoll := 801.0);
   Bridle_04 : UDT_Bridle_3M := (PF755_shaft_a.DL_In.PTP_Feedback := 1828521382, PF755_shaft_a.DL_In.P7_Ptc_Sts := 1, PF755_shaft_a.DL_In.P7_DigitalInSts := 2#0000_0000_0000_0000_0000_0000_0000_0011, PF755_shaft_a.IO_ConnectionOk := 1, PF755_shaft_b.DL_In.PTP_Feedback := 7917204, PF755_shaft_b.DL_In.P7_Ptc_Sts := 1, PF755_shaft_b.DL_In.P7_DigitalInSts := 2#0000_0000_0000_0000_0000_0000_0000_0011, PF755_shaft_b.IO_ConnectionOk := 1, PF755_shaft_c.DL_In.PTP_Feedback := 769240356, PF755_shaft_c.DL_In.P7_Ptc_Sts := 4, PF755_shaft_c.DL_In.P7_DigitalInSts := 2#0000_0000_0000_0000_0000_0000_0000_0011, PF755_shaft_c.IO_ConnectionOk := 1, Stat.Stopped := 1, Stat.AllEnabled := 1, Stat.AllStandStill := 1, Stat.All_CB_Ok := 1, Stat.AllSafetyOk := 1, Stat.NoFastStop := 1, Stat.NoPrecharge := 1, Stat.AllReady := 1, Stat.NoOverTemp := 1, Stat.IOConnOkAllDrvs := 1, Config_shaft_a.zGearRatio := 138.56, Config_shaft_a.DiameterRoll := 801.0, Config_shaft_b.zGearRatio := 129.41, Config_shaft_b.DiameterRoll := 801.0, Config_shaft_c.zGearRatio := 27.88, Config_shaft_c.DiameterRoll := 200.0);
   Bridle_04_FB_Diff : DINT;
   Bridle_04_FB_Update_Valid : BOOL;
   Bridle_04_Rev_mm : REAL := 0.05142632;
   Bridle_04b_FBCounts_mm : REAL := 210.64221;
   comm_mw : DINT[15];
   cu : UDT_Pinchroll := (PF755.DL_In.OutputVoltage := 1.2345252e-20, PF755.DL_In.P7_Ptc_Sts := 4, PF755.DL_In.P7_DigitalInSts := 2#0000_0000_0000_0000_0000_0000_0000_0011, PF755.DL_Out.SpdRegNegLim := -30.0, PF755.DL_Out.SpdRegPosLim := 30.0, PF755.IO_ConnectionOk := 1, PF755.Reference := 3.803062, Cmd.MtrCb := 1, Stat.Stopped := 1, Stat.CB_Ok := 1, Stat.SafetyOk := 1, Stat.NoFastStop := 1, Stat.NoPrecharge := 1, Stat.Ready := 1, Stat.NoOverTemp := 1, Config.zGearRatio := 15.0, Config.DiameterRoll := 250.0, Config.zMaxAcc := 0.1, Config.zMaxDec := 0.1, Config.zJogRef := 0.1, Config.zAccJog := 0.2, Config.zDecJog := 0.2, Config.zJerkJog := 0.2);
   Entry_Accu : UDT_Entry_Accu := (PF755.DL_In.OutputFrequency := 0.018556317, PF755.DL_In.OutputCurrent := 32.354126, PF755.DL_In.OutputVoltage := 4.604002, PF755.DL_In.OutputPower := 0.25720245, PF755.DL_In.SRegOutput := 3.001518, PF755.DL_In.PTP_Feedback := 6033754, PF755.DL_In.LimitedTrqRef := 3.001518, PF755.DL_In.P7_Ptc_Sts := 1, PF755.DL_In.P7_DigitalOutSts := 3, PF755.DL_In.P7_DigitalInSts := 2#0000_0000_0000_0000_0000_0000_0000_0111, PF755.DL_In.HomingStatus := 8, PF755.DL_Out.TorqueSp := -1.2e-43, PF755.DL_Out.RegulatorMode := -198601572, PF755.DL_Out.UserHomePos := 8252524, PF755.DL_Out.SpdRegNegLim := -50.0, PF755.DL_Out.SpdRegPosLim := 50.0, PF755.IO_ConnectionOk := 1, PF755.Reference := -0.0041867304, Cmd.Run := 1, Stat.Held := 1, Stat.BrOk := 1, Stat.CB_Ok := 1, Stat.SafetyOk := 1, Stat.NoFastStop := 1, Stat.NoPrecharge := 1, Stat.Ready := 1, Stat.NoOverTemp := 1, Stat.FanOn := 1, Stat.Synch := 1, Stat.TenRegOnSp := 1, Stat.NotAtLimit := 1, Fdbk.PvActualPos := 8131.7437, Fdbk.PvActualPosPct := 69.680756, Fdbk.PvSpdRef_MPS := -3.853056e-07, Fdbk.PvSpdRef_RPM := -0.0041867304, Sp.SpPos := 93.0, Config.zGearRatio := 0.1811, Config.zMaxPos := 11670.0, Config.zSyncPos := 11122.0, Config.zJogRef := 0.02, Config.zAccJog := 0.04, Config.zDecJog := 0.04, Config.zJerkJog := 0.25, Ctrl.Run := 1, Ctrl.URmpdRefEnable := 1, Ctrl.TenRegOn := 1, Ctrl.SpdTrim := 0.00017210045);
   Entry_Drives_StandStill : BOOL;
   EntryAccuMatLgth : REAL := 15320.291;
   EntryCmd : UDT_Commands_Zone;
   EntryConfig : UDT_Config_Zone := (zJogRef := 0.1, zAccJog := 0.083, zDecJog := 0.083, zJerkJog := 0.1, zAccRun := 0.04, zDecRun := 0.04, zJerkRun := 0.15, zMaxAccDec := 0.25, zMaxSpd := 0.5);
   EntryCtrl : UDT_Control_Zone;
   EntryFdbks : UDT_Feedbacks_Zone;
   EntrySetpoints : UDT_Setpoints_Zone;
   EntryStat : UDT_Status_Zone := (AllDrivesEnabled := 1, IOConnOkDrives := 1, NoFastStop := 1, SafetyOkAllDrvs := 1, AllDrivesAtZeroSpd := 1, DrivesReady := 1, Standstilll := 1, BR_Ok := 1, All_CB_Ok := 1, Ready := 1);
   Exit_Accu : UDT_Exit_Accu := (PF755.DL_In.OutputFrequency := 0.07859213, PF755.DL_In.OutputCurrent := 36.02611, PF755.DL_In.OutputVoltage := 5.686399, PF755.DL_In.OutputPower := 0.34736156, PF755.DL_In.SRegOutput := 11.088152, PF755.DL_In.PTP_Feedback := 1565812, PF755.DL_In.LimitedTrqRef := 11.088152, PF755.DL_In.P7_Ptc_Sts := 1, PF755.DL_In.P7_DigitalOutSts := 3, PF755.DL_In.P7_DigitalInSts := 2#0000_0000_0000_0000_0000_0000_0000_0111, PF755.DL_In.HomingStatus := 8, PF755.DL_Out.UserHomePos := 298570, PF755.DL_Out.SpdRegNegLim := -50.0, PF755.DL_Out.SpdRegPosLim := 50.0, PF755.IO_ConnectionOk := 1, PF755.Feedback := 0.3499273, PF755.Reference := 0.23410717, Cmd.Run := 1, Stat.Held := 1, Stat.BrOk := 1, Stat.CB_Ok := 1, Stat.SafetyOk := 1, Stat.NoFastStop := 1, Stat.NoPrecharge := 1, Stat.Ready := 1, Stat.NoOverTemp := 1, Stat.FanOn := 1, Stat.Synch := 1, Stat.TenRegOnSp := 1, Stat.NotAtLimit := 1, Fdbk.PvSpeed := 0.031143531, Fdbk.PvActualPos := 4289.8955, Fdbk.PvActualPosPct := 14.626307, Fdbk.PvSpdRef_MPS := 4.3840293e-05, Fdbk.PvSpdRef_RPM := 0.23410717, Sp.SpPos := 5.0, Config.zGearRatio := 0.089, Config.zMaxPos := 29330.0, Config.zSyncPos := 818.0, Config.zJogRef := 0.041, Config.zAccJog := 0.08, Config.zDecJog := 0.08, Config.zJerkJog := 0.25, Ctrl.Run := 1, Ctrl.URmpdRefEnable := 1, Ctrl.TenRegOn := 1, Ctrl.SpdTrim := -0.00030113122);
   Exit_Accu_RdfnPos : TIMER := (PRE := 600);
   Exit_Drives_StandStill : BOOL;
   Exit_PosSp_AtShear : DINT := 100;
   Exit_PosSp_ToWinder : DINT := 100;
   ExitCmd : UDT_Commands_Zone;
   ExitConfig : UDT_Config_Zone := (zJogRef := 0.116, zAccJog := 0.083, zDecJog := 0.083, zJerkJog := 0.25, zAccRun := 0.04, zDecRun := 0.04, zJerkRun := 0.15, zMaxAccDec := 0.25, zMaxSpd := 0.5);
   ExitCtrl : UDT_Control_Zone;
   ExitFdbks : UDT_Feedbacks_Zone := (PvSpeedRef := 0.13333334);
   ExitSetpoints : UDT_Setpoints_Zone;
   ExitStat : UDT_Status_Zone := (AllDrivesEnabled := 1, IOConnOkDrives := 1, NoFastStop := 1, SafetyOkAllDrvs := 1, DrivesReady := 1, Standstilll := 1, BR_Ok := 1, All_CB_Ok := 1, Ready := 1);
   ForSimulation : REAL[100];
   In_Commands : UDT_Commands := (Line.WD_FromMaster := 1, Entry_Accu.Run := 1, Exit_Accu.Run := 1, cu.MtrCb := 1);
   In_Config : UDT_Config;
   In_Setpoints : UDT_Setpoints := (Unwinder_1.SpNewDiameter := 800.0, Unwinder_1.SpTension := 9950.0, Unwinder_1.zCellToStitch := 1500.0, Unwinder_1.zCellToShear := 1000.0, Unwinder_2.SpNewDiameter := 800.0, Unwinder_2.SpTension := 6500.0, Unwinder_2.zCellToStitch := 1500.0, Unwinder_2.zCellToShear := 1000.0, Entry_Accu.SpPos := 93.0, Exit_Accu.SpPos := 5.0, Winder.SpNewDiameter := 600.0, Winder.SpTension := 10000.0, Winder.zCellToStitch := 3000.0, Winder.zCellToShear := 3200.0, TM1.SpTen := 5850.0, TM1.PvTen := 5850.0, TM1.MaxTen := 30000.0, TM2.SpTen := 8250.0, TM2.PvTen := 1830.0, TM2.MaxTen := 50000.0, TM3.SpTen := 6900.0, TM3.PvTen := 6840.0, TM3.MaxTen := 50000.0, Line.WebWidth := 500.0, Line.MaterialDensity := 3725.0, Line.SpMmPerRev := 25.0, Line.JogSpdRef := 0.083);
   LineCmd : UDT_Commands_Line;
   LineConfig : UDT_Config_Line := (zAccRate := 0.04, zDecRate := 0.04, zJerk := 0.15, zJogSpd := 0.1, zJogAccRate := 0.083, zJogDecRate := 0.083, zMaxAccDec := 0.25, zSpdMax := 0.25);
   LineCtrl : UDT_Control_Line := (SpdRefRmp := 0.00068994303);
   LineFdbks : UDT_Feedbacks_Line := (Stitch_Cntrs.Zone_2[0] := 134239.52);
   LineSetpoints : UDT_Setpoints_Line := (WebWidth := 500.0, MaterialDensity := 3725.0, SpMmPerRev := 25.0, JogSpdRef := 0.083);
   LineStat : UDT_Status_Line := (WD_ToMaster := 1, MasterPlcOk := 1, DrivesReady := 1, LineReady := 1, NoFastStop := 1, AllStandstill := 1);
   MainFltHndler : DINT[11];
   nbrstiychout : DINT := 8123;
   offst_pr_br1 : REAL := 0.2;
   Out_Feedbacks : UDT_Fdbks := (Unwinder_1.PvActualDiameter := 547.79364, Unwinder_1.PvNormInertia := 2.0793295, Unwinder_1.PvTotalInertia := 1.0057888, Unwinder_1.PvCoilLength := 7613.1245, Unwinder_2.PvActualDiameter := 563.14075, Unwinder_2.PvNormInertia := 2.080902, Unwinder_2.PvTotalInertia := 1.0065495, Unwinder_2.PvCoilLength := 194935.27, Entry_Accu.PvActualPos := 8131.7437, Entry_Accu.PvActualPosPct := 69.680756, Entry_Accu.PvSpdRef_MPS := -3.853056e-07, Entry_Accu.PvSpdRef_RPM := -0.0041867304, Bridle_02a.SpSpdRef_MPS := 0.00068994303, Bridle_02b.SpSpdRef_MPS := 0.00068994303, Bridle_03a.SpSpdRef_MPS := 0.00068994303, Bridle_03b.SpSpdRef_MPS := 0.00068994303, Exit_Accu.PvSpeed := 0.035492375, Exit_Accu.PvActualPos := 4290.1587, Exit_Accu.PvActualPosPct := 14.627203, Exit_Accu.PvSpdRef_MPS := 7.314191e-05, Exit_Accu.PvSpdRef_RPM := 0.39057782, Pinchroll_3.PvSpdRef_RPM := nan, Winder.PvActualDiameter := 709.3403, Winder.PvNormInertia := 0.79611427, Winder.PvTotalInertia := 1.0009869, Winder.PvCoilLength := 143400.64, Line.Stitch_Cntrs.Zone_2[0] := 134239.52, Exit.PvSpeedRef := 0.13333334); {produced}
   Out_Status : UDT_Status := (Line.MasterPlcOk := 1, Line.DrivesReady := 1, Line.LineReady := 1, Line.NoFastStop := 1, Line.AllStandstill := 1, Entry.AllDrivesEnabled := 1, Entry.IOConnOkDrives := 1, Entry.NoFastStop := 1, Entry.SafetyOkAllDrvs := 1, Entry.AllDrivesAtZeroSpd := 1, Entry.DrivesReady := 1, Entry.Standstilll := 1, Entry.BR_Ok := 1, Entry.All_CB_Ok := 1, Entry.Ready := 1, Exit.AllDrivesEnabled := 1, Exit.IOConnOkDrives := 1, Exit.NoFastStop := 1, Exit.SafetyOkAllDrvs := 1, Exit.DrivesReady := 1, Exit.Standstilll := 1, Exit.BR_Ok := 1, Exit.All_CB_Ok := 1, Exit.Ready := 1, Unwinder_1.Stopped := 1, Unwinder_1.CB_Ok := 1, Unwinder_1.SafetyOk := 1, Unwinder_1.NoFastStop := 1, Unwinder_1.NoPrecharge := 1, Unwinder_1.Ready := 1, Unwinder_1.NoOverTemp := 1, Unwinder_2.Stopped := 1, Unwinder_2.CB_Ok := 1, Unwinder_2.SafetyOk := 1, Unwinder_2.NoFastStop := 1, Unwinder_2.NoPrecharge := 1, Unwinder_2.Ready := 1, Unwinder_2.NoOverTemp := 1, Pinchroll_1.Stopped := 1, Pinchroll_1.CB_Ok := 1, Pinchroll_1.SafetyOk := 1, Pinchroll_1.NoFastStop := 1, Pinchroll_1.NoPrecharge := 1, Pinchroll_1.Ready := 1, Pinchroll_1.NoOverTemp := 1, Pinchroll_2.Stopped := 1, Pinchroll_2.CB_Ok := 1, Pinchroll_2.SafetyOk := 1, Pinchroll_2.NoFastStop := 1, Pinchroll_2.NoPrecharge := 1, Pinchroll_2.Ready := 1, Pinchroll_2.NoOverTemp := 1, Entry_Accu.Held := 1, Entry_Accu.BrOk := 1, Entry_Accu.CB_Ok := 1, Entry_Accu.SafetyOk := 1, Entry_Accu.NoFastStop := 1, Entry_Accu.NoPrecharge := 1, Entry_Accu.Ready := 1, Entry_Accu.NoOverTemp := 1,
        Entry_Accu.FanOn := 1, Entry_Accu.Synch := 1, Entry_Accu.TenRegOnSp := 1, Entry_Accu.NotAtLimit := 1, Bridle_01.Stopped := 1, Bridle_01.AllEnabled := 1, Bridle_01.AllStandStill := 1, Bridle_01.All_CB_Ok := 1, Bridle_01.AllSafetyOk := 1, Bridle_01.NoFastStop := 1, Bridle_01.NoPrecharge := 1, Bridle_01.AllReady := 1, Bridle_01.NoOverTemp := 1, Bridle_01.IOConnOkAllDrvs := 1, Bridle_02.Stopped := 1, Bridle_02.AllEnabled := 1, Bridle_02.AllStandStill := 1, Bridle_02.All_CB_Ok := 1, Bridle_02.AllSafetyOk := 1, Bridle_02.NoFastStop := 1, Bridle_02.NoPrecharge := 1, Bridle_02.AllReady := 1, Bridle_02.NoOverTemp := 1, Bridle_02.IOConnOkAllDrvs := 1, Bridle_03.Stopped := 1, Bridle_03.AllEnabled := 1, Bridle_03.AllStandStill := 1, Bridle_03.All_CB_Ok := 1, Bridle_03.AllSafetyOk := 1, Bridle_03.NoFastStop := 1, Bridle_03.NoPrecharge := 1, Bridle_03.AllReady := 1, Bridle_03.NoOverTemp := 1, Bridle_03.IOConnOkAllDrvs := 1, Bridle_04.Stopped := 1, Bridle_04.AllEnabled := 1, Bridle_04.AllStandStill := 1, Bridle_04.All_CB_Ok := 1, Bridle_04.AllSafetyOk := 1, Bridle_04.NoFastStop := 1, Bridle_04.NoPrecharge := 1, Bridle_04.AllReady := 1, Bridle_04.NoOverTemp := 1, Bridle_04.IOConnOkAllDrvs := 1, Exit_Accu.Held := 1, Exit_Accu.BrOk := 1, Exit_Accu.CB_Ok := 1, Exit_Accu.SafetyOk := 1, Exit_Accu.NoFastStop := 1, Exit_Accu.NoPrecharge := 1, Exit_Accu.Ready := 1, Exit_Accu.NoOverTemp := 1, Exit_Accu.FanOn := 1, Exit_Accu.Synch := 1, Exit_Accu.TenRegOnSp := 1, Exit_Accu.NotAtLimit := 1, Pinchroll_3.SafetyOk := 1, Pinchroll_3.NoPrecharge := 1, Pinchroll_3.Ready := 1, Pinchroll_3.NoOverTemp := 1,
        Winder.Stopped := 1, Winder.CB_Ok := 1, Winder.SafetyOk := 1, Winder.NoFastStop := 1, Winder.NoPrecharge := 1, Winder.Ready := 1, Winder.NoOverTemp := 1, cu.Stopped := 1, cu.CB_Ok := 1, cu.SafetyOk := 1, cu.NoFastStop := 1, cu.NoPrecharge := 1, cu.Ready := 1, cu.NoOverTemp := 1); {produced}
   par_winder_JAR : REAL := 0.87;
   Pinchroll_1 : UDT_Pinchroll := (PF755.DL_In.PTP_Feedback := 34142675, PF755.DL_In.P7_Ptc_Sts := 1, PF755.DL_In.P7_DigitalInSts := 2#0000_0000_0000_0000_0000_0000_0000_0011, PF755.IO_ConnectionOk := 1, Stat.Stopped := 1, Stat.CB_Ok := 1, Stat.SafetyOk := 1, Stat.NoFastStop := 1, Stat.NoPrecharge := 1, Stat.Ready := 1, Stat.NoOverTemp := 1, Config.zGearRatio := 33.0, Config.DiameterRoll := 491.0, Config.zMaxAcc := 0.1, Config.zMaxDec := 0.1, Config.zJogRef := 0.083, Config.zAccJog := 0.16, Config.zDecJog := 0.16, Config.zJerkJog := 0.25);
   Pinchroll_2 : UDT_Pinchroll := (PF755.DL_In.PTP_Feedback := 372815085, PF755.DL_In.P7_Ptc_Sts := 1, PF755.DL_In.P7_DigitalInSts := 2#0000_0000_0000_0000_0000_0000_0000_0011, PF755.IO_ConnectionOk := 1, Stat.Stopped := 1, Stat.CB_Ok := 1, Stat.SafetyOk := 1, Stat.NoFastStop := 1, Stat.NoPrecharge := 1, Stat.Ready := 1, Stat.NoOverTemp := 1, Config.zGearRatio := 97.0, Config.DiameterRoll := 582.25, Config.zMaxAcc := 0.1, Config.zMaxDec := 0.1, Config.zJogRef := 0.083, Config.zAccJog := 0.16, Config.zDecJog := 0.16, Config.zJerkJog := 0.25);
   Pinchroll_2_FB_Difference : DINT;
   Pinchroll_2_FB_Update_Valid : BOOL;
   Pinchroll_2_FBCounts_mm : REAL := 217.20624;
   Pinchroll_3 : UDT_Pinchroll := (PF755.DL_In.P7_DigitalInSts := 2#0000_0000_0000_0000_0000_0000_0000_0001, PF755.IO_ConnectionOk := 1, Stat.Held := 1, Stat.SafetyOk := 1, Stat.NoPrecharge := 1, Stat.Ready := 1, Stat.NoOverTemp := 1, Config.zGearRatio := 15.0, Config.DiameterRoll := 250.0, Config.zMaxAcc := 0.1, Config.zMaxDec := 0.1, Config.zJogRef := 0.1, Config.zAccJog := 0.2, Config.zDecJog := 0.2, Config.zJerkJog := 0.2);
   Pinchroll_3_FB_Diff : DINT;
   Pinchroll_3_FB_Update_Valid : BOOL;
   Pinchroll_3_FBCounts_mm : DINT := 20;
   Pinchroll_3_Max_FB_Counts : DINT := 1280;
   Pinchroll_3_Rev_mm : REAL := 0.019098593;
   Stitch_Cntrs : UDT_Stitch_Counter := (Zone_2[0] := 134239.52);
   TaskInterval_micro_sec : DINT := 50000;
   TaskInterval_ms : DINT := 50;
   TblStitchVal : UDT_Stitch_Counter[10];
   TestCmdBridle_02 : UDT_Commands_Bridle := (JogFwd := 1);
   TestCmdBridle_03 : UDT_Commands_Bridle;
   TestConfig_Bridle_01a : UDT_Config_Bridle := (zGearRatio := 129.41, DiameterRoll := 801.0);
   TestConfig_Bridle_01b : UDT_Config_Bridle := (zGearRatio := 129.41, DiameterRoll := 801.0);
   TestConfig_Bridle_01c : UDT_Config_Bridle := (zGearRatio := 27.88, DiameterRoll := 202.12);
   TestConfig_Bridle_02a : UDT_Config_Bridle := (zGearRatio := 256.39, DiameterRoll := 801.0);
   TestConfig_Bridle_02b : UDT_Config_Bridle := (zGearRatio := 256.39, DiameterRoll := 801.0);
   TestConfig_Bridle_03a : UDT_Config_Bridle := (zGearRatio := 256.39, DiameterRoll := 801.0);
   TestConfig_Bridle_03b : UDT_Config_Bridle := (zGearRatio := 256.39, DiameterRoll := 801.0);
   TestConfig_Bridle_04a : UDT_Config_Bridle := (zGearRatio := 138.56, DiameterRoll := 801.0);
   TestConfig_Bridle_04b : UDT_Config_Bridle := (zGearRatio := 129.41, DiameterRoll := 801.0);
   TestConfig_Bridle_04c : UDT_Config_Bridle := (zGearRatio := 27.88, DiameterRoll := 200.0);
   TestConfig_cu : UDT_Config_Pinch := (zGearRatio := 199.0, DiameterRoll := 689.5, zMaxAcc := 0.5, zMaxDec := 0.5, zJogRef := 0.233, zAccJog := 0.16, zDecJog := 0.16, zJerkJog := 0.25);
   TestConfig_Entry : UDT_Config_Zone := (zJogRef := 0.1, zAccJog := 0.083, zDecJog := 0.083, zJerkJog := 0.1, zAccRun := 0.04, zDecRun := 0.04, zJerkRun := 0.15, zMaxAccDec := 0.25, zMaxSpd := 0.5);
   TestConfig_Entry_Accu : UDT_Config_Accu := (zGearRatio := 0.1811, zMaxPos := 11670.0, zSyncPos := 11122.0, zJogRef := 0.02, zAccJog := 0.04, zDecJog := 0.04, zJerkJog := 0.25);
   TestConfig_Exit : UDT_Config_Zone := (zJogRef := 0.116, zAccJog := 0.083, zDecJog := 0.083, zJerkJog := 0.25, zAccRun := 0.04, zDecRun := 0.04, zJerkRun := 0.15, zMaxAccDec := 0.25, zMaxSpd := 0.5);
   TestConfig_Exit_Accu : UDT_Config_Accu := (zGearRatio := 0.089, zMaxPos := 29330.0, zSyncPos := 818.0, zJogRef := 0.041, zAccJog := 0.08, zDecJog := 0.08, zJerkJog := 0.25);
   TestConfig_Line : UDT_Config_Line := (zAccRate := 0.04, zDecRate := 0.04, zJerk := 0.15, zJogSpd := 0.1, zJogAccRate := 0.083, zJogDecRate := 0.083, zMaxAccDec := 0.25, zSpdMax := 0.25);
   TestConfig_Pinchroll_1 : UDT_Config_Pinch := (zGearRatio := 33.0, DiameterRoll := 491.0, zMaxAcc := 0.1, zMaxDec := 0.1, zJogRef := 0.083, zAccJog := 0.16, zDecJog := 0.16, zJerkJog := 0.25);
   TestConfig_Pinchroll_2 : UDT_Config_Pinch := (zGearRatio := 97.0, DiameterRoll := 582.25, zMaxAcc := 0.1, zMaxDec := 0.1, zJogRef := 0.083, zAccJog := 0.16, zDecJog := 0.16, zJerkJog := 0.25);
   TestConfig_Pinchroll_3 : UDT_Config_Pinch := (zGearRatio := 15.0, DiameterRoll := 250.0, zMaxAcc := 0.5, zMaxDec := 0.5, zJogRef := 0.083, zAccJog := 0.16, zDecJog := 0.16, zJerkJog := 0.25);
   TestConfig_Unwinder_1 : UDT_Config_Unwinder := (zGearRatio := 78.0, zMinDiameter := 500.0, zMaxDiameter := 2000.0, zMaxTension := 15000.0, zJogRef := 0.083, zDiamCalcEnblThresh_MPS := 1.e-04, zDiamCalcUpdate_Rev := 0.5, zMotorPwr := 11.0, zMtrBaseSpd := 1440.0, zAccJog := 0.16, zDecJog := 0.16, zJerkJog := 0.25);
   TestConfig_Unwinder_2 : UDT_Config_Unwinder := (zGearRatio := 78.0, zMinDiameter := 500.0, zMaxDiameter := 2000.0, zMinTension := 1.0, zMaxTension := 15000.0, zJogRef := 0.083, zDiamCalcEnblThresh_MPS := 1.e-04, zDiamCalcUpdate_Rev := 0.5, zMotorPwr := 11.0, zMtrBaseSpd := 1440.0, zAccJog := 0.16, zDecJog := 0.16, zJerkJog := 0.25);
   TestConfig_Winder : UDT_Config_Unwinder := (zGearRatio := 268.0, zMinDiameter := 508.0, zMaxDiameter := 2000.0, zMinTension := 1.0, zMaxTension := 50000.0, zJogRef := 0.13, zDiamCalcEnblThresh_MPS := 1.e-04, zDiamCalcUpdate_Rev := 0.5, zMotorPwr := 30.0, zMtrBaseSpd := 1475.0, zAccJog := 0.1, zDecJog := 0.25, zJerkJog := 0.5);
   TestSp_Entry : UDT_Setpoints_Zone := (MaxSpdRef := 0.1);
   TestSp_Entry_Accu : UDT_Setpoints_Accu := (SpPos := 60.0);
   TestSp_Exit : UDT_Setpoints_Zone := (MaxSpdRef := 0.1);
   TestSp_Exit_Accu : UDT_Setpoints_Accu := (SpPos := 10.0);
   TestSp_Line : UDT_Setpoints_Line := (RunSpdRef := 0.1, WebWidth := 1250.0, MaterialDensity := 3725.0, SpMmPerRev := 25.0, JogSpdRef := 0.083);
   TestSp_TM1 : UDT_Setpoints_TM := (SpTen := 250.0, MaxTen := 1000.0);
   TestSp_TM2 : UDT_Setpoints_TM := (SpTen := 250.0, MaxTen := 1000.0);
   TestSp_TM3 : UDT_Setpoints_TM := (SpTen := 250.0, MaxTen := 1000.0);
   TestSp_Unwinder_1 : UDT_Setpoints_Unwinder := (SpNewDiameter := 250.0, SpTension := 50.0);
   TestSp_Unwinder_2 : UDT_Setpoints_Unwinder := (SpNewDiameter := 1500.0, SpTension := 1000.0);
   TestSp_Winder : UDT_Setpoints_Unwinder := (SpNewDiameter := 508.0, SpTension := 100.0, zCellToStitch := 1500.0, zCellToShear := 5000.0);
   TM1 : UDT_TM := (Sp.SpTen := 5850.0, Sp.PvTen := 5840.0, Sp.MaxTen := 30000.0);
   TM2 : UDT_TM := (Sp.SpTen := 8250.0, Sp.PvTen := 1850.0, Sp.MaxTen := 50000.0);
   TM3 : UDT_TM := (Sp.SpTen := 6900.0, Sp.PvTen := 6890.0, Sp.MaxTen := 50000.0);
   Unwinder_1 : UDT_Unwinder := (PF755.DL_In.PTP_Feedback := -2135218541, PF755.DL_In.P7_Ptc_Sts := 4, PF755.DL_In.P7_DigitalInSts := 2#0000_0000_0000_0000_0000_0000_0000_0011, PF755.DL_Out.RegulatorMode := 1, PF755.DL_Out.SpeedRegBW := 25.87539, PF755.IO_ConnectionOk := 1, Stat.Stopped := 1, Stat.CB_Ok := 1, Stat.SafetyOk := 1, Stat.NoFastStop := 1, Stat.NoPrecharge := 1, Stat.Ready := 1, Stat.NoOverTemp := 1, Fdbk.PvActualDiameter := 547.79364, Fdbk.PvNormInertia := 2.0793295, Fdbk.PvTotalInertia := 1.0057888, Fdbk.PvCoilLength := 7613.1245, Sp.SpNewDiameter := 800.0, Sp.SpTension := 9950.0, Sp.zCellToStitch := 1500.0, Sp.zCellToShear := 1000.0, Config.zGearRatio := 78.0, Config.zMinDiameter := 500.0, Config.zMaxDiameter := 2000.0, Config.zMaxTension := 15000.0, Config.zJogRef := 0.083, Config.zDiamCalcEnblThresh_MPS := 1.e-04, Config.zDiamCalcUpdate_Rev := 0.5, Config.zMotorPwr := 11.0, Config.zMtrBaseSpd := 1440.0, Config.zAccJog := 0.16, Config.zDecJog := 0.16, Config.zJerkJog := 0.25);
   Unwinder_2 : UDT_Unwinder := (PF755.DL_In.PTP_Feedback := 1613409681, PF755.DL_In.P7_Ptc_Sts := 4, PF755.DL_In.P7_DigitalInSts := 2#0000_0000_0000_0000_0000_0000_0000_0011, PF755.DL_Out.RegulatorMode := 1, PF755.DL_Out.SpeedRegBW := 25.960638, PF755.IO_ConnectionOk := 1, Stat.Stopped := 1, Stat.CB_Ok := 1, Stat.SafetyOk := 1, Stat.NoFastStop := 1, Stat.NoPrecharge := 1, Stat.Ready := 1, Stat.NoOverTemp := 1, Fdbk.PvActualDiameter := 563.14075, Fdbk.PvNormInertia := 2.080902, Fdbk.PvTotalInertia := 1.0065495, Fdbk.PvCoilLength := 194935.27, Sp.SpNewDiameter := 800.0, Sp.SpTension := 6500.0, Sp.zCellToStitch := 1500.0, Sp.zCellToShear := 1000.0, Config.zGearRatio := 78.0, Config.zMinDiameter := 500.0, Config.zMaxDiameter := 2000.0, Config.zMinTension := 1.0, Config.zMaxTension := 15000.0, Config.zJogRef := 0.083, Config.zDiamCalcEnblThresh_MPS := 1.e-04, Config.zDiamCalcUpdate_Rev := 0.5, Config.zMotorPwr := 11.0, Config.zMtrBaseSpd := 1440.0, Config.zAccJog := 0.16, Config.zDecJog := 0.16, Config.zJerkJog := 0.25);
   ValWindowMin : REAL := 17820.291;
   voirmw : BOOL;
   Winder : UDT_Winder := (PF755.DL_In.PTP_Feedback := -561673658, PF755.DL_In.P7_Ptc_Sts := 1, PF755.DL_In.P7_DigitalInSts := 2#0000_0000_0000_0000_0000_0000_0000_0111, PF755.DL_Out.RegulatorMode := 1, PF755.DL_Out.SpeedRegBW := 35.0, PF755.IO_ConnectionOk := 1, Stat.Stopped := 1, Stat.CB_Ok := 1, Stat.SafetyOk := 1, Stat.NoFastStop := 1, Stat.NoPrecharge := 1, Stat.Ready := 1, Stat.NoOverTemp := 1, Fdbk.PvActualDiameter := 709.3403, Fdbk.PvNormInertia := 0.79611427, Fdbk.PvTotalInertia := 1.0009869, Fdbk.PvCoilLength := 143400.64, Sp.SpNewDiameter := 600.0, Sp.SpTension := 10000.0, Sp.zCellToStitch := 3000.0, Sp.zCellToShear := 3200.0, Config.zGearRatio := 268.0, Config.zMinDiameter := 508.0, Config.zMaxDiameter := 2000.0, Config.zMinTension := 1.0, Config.zMaxTension := 50000.0, Config.zJogRef := 0.13, Config.zDiamCalcEnblThresh_MPS := 1.e-04, Config.zDiamCalcUpdate_Rev := 0.5, Config.zMotorPwr := 30.0, Config.zMtrBaseSpd := 1475.0, Config.zAccJog := 0.1, Config.zDecJog := 0.25, Config.zJerkJog := 0.5);
   Winder_FB_Counts_Diff : DINT;
   Winder_FB_Counts_mm : DINT := 493;
   Winder_FB_Update_Valid : BOOL;
   zBridle_01a_EncRes : DINT := 4096;
   zBridle_02a_EncRes : DINT := 4096;
   zBridle_03a_EncRes : DINT := 4096;
   zBridle_04a_EncRes : DINT := 4096;
   zBridle_04b_Max_rev : REAL := 1500.0;
   zConfigFromMaster : BOOL;
   zCuSpdTrimMltp : REAL := 0.2;
   zEntryAccuLngthOffs : REAL := 8050.0;
   zExit_Accu_NrOfCyl : DINT := 2;
   zExit_Dist_ShearToWinder : DINT := 100;
   zNoMaster : BOOL := 1;
   zPi : REAL := 3.1415927; {constant, access Read Only}
   zPinchroll_2_EncRes : DINT := 4096;
   zPinchroll_3_EncRes : DINT := 4096;
   zSimulation : BOOL; {access Read Only}
   zStitcherToAccu : REAL := 17000.0;
   zStitchValOffset : REAL := 250.0;
   zWinderDiamFullTrq : REAL := 1000.0;
END_VAR

PROGRAM P00_Line   (* main routine R00_Main *)
VAR
   ArrSize_Z1 : DINT := 3;
   ArrSize_Z2 : DINT := 5;
   BAND_01 : FBD_BOOLEAN_AND := (In3 := 1, In4 := 1, In5 := 1, In6 := 1, In7 := 1, In8 := 1);
   BAND_02 : FBD_BOOLEAN_AND := (In3 := 1, In4 := 1, In5 := 1, In6 := 1, In7 := 1, In8 := 1);
   BAND_03 : FBD_BOOLEAN_AND := (In3 := 1, In4 := 1, In5 := 1, In6 := 1, In7 := 1, In8 := 1);
   BNOT_01 : FBD_BOOLEAN_NOT := (Out := 1);
   BOR_02 : FBD_BOOLEAN_OR;
   BOR_03 : FBD_BOOLEAN_OR;
   Bridle_01_MM_Count : REAL := 0.0047473866;
   Bridle_02_MM_Count : REAL := 0.0023584906;
   Bridle_04_MM_Count : REAL := 0.0047473866;
   Entry_Accu_Mat_Length : DINT := 32527;
   Exit_Accu_Mat_Length : REAL := 8581.276;
   HLL_01 : HL_LIMIT := (HighLimit := 0.25, LowLimit := -0.25);
   Indexer : DINT;
   NEG_01 : FBD_MATH_ADVANCED := (Source := 0.083, Dest := -0.083);
   NEG_02 : FBD_MATH_ADVANCED := (Source := 0.25, Dest := -0.25);
   NewStitch_Z1_ons : FBD_ONESHOT;
   NewStitch_Z2_Ons : FBD_ONESHOT;
   NewStitch_Z3_Ons : FBD_ONESHOT;
   NrStitch_Z1 : DINT;
   NrStitch_Z2 : DINT := 1;
   Ons : BOOL[32] := ([3] := 1);
   Preset_Max_Z2 : REAL[5] := ([0] := 197358.14);
   RLIM_01 : RATE_LIMITER := (In := 0.00068994303, IncRate := 0.25, DecRate := 0.25, RTSTime := 1, Out := 0.00068994303, DeltaT := 0.05);
   SCRV_01 : S_CURVE := (JerkRate := 0.15, RTSTime := 1, Out := 0.00068994303, DeltaT := 0.05);
   SEL_01 : SELECT;
   SSUM_01 : SELECTED_SUMMER := (Gain1 := 1.0, In2 := 0.083, Gain2 := 1.0, Gain3 := 1.0, Select3 := 1, In4 := -0.083, Gain4 := 1.0, Gain5 := 1.0, Gain6 := 1.0, Gain7 := 1.0, Gain8 := 1.0);
   SSUM_03 : SELECTED_SUMMER := (In1 := 0.04, Gain1 := 1.0, In2 := 0.083, Gain2 := 1.0, Gain3 := 1.0, Gain4 := 1.0, Gain5 := 1.0, Gain6 := 1.0, Gain7 := 1.0, Gain8 := 1.0);
   SSUM_04 : SELECTED_SUMMER := (In1 := 0.04, Gain1 := 1.0, In2 := 0.083, Gain2 := 1.0, Gain3 := 1.0, Gain4 := 1.0, Gain5 := 1.0, Gain6 := 1.0, Gain7 := 1.0, Gain8 := 1.0);
   StitchIn_Z1 : BOOL;
   StitchIn_Z2 : BOOL;
   StitchIn_Z3 : BOOL;
   StitchValMin : REAL := -15500.0;
   StitchValPlus : REAL := 15500.0;
   TofStitch_Z2 : TIMER := (PRE := 1000, ACC := 1000);
   TofStitch_Z3 : TIMER := (PRE := 1000, ACC := 1000);
   TofWatchDogMaster : TIMER := (PRE := 1000, EN := 1, DN := 1);
   Update_Cntrs_Z1 : BOOL;
   Update_Cntrs_Z2 : BOOL;
   ValCntrs_Z2 : REAL[5] := ([0] := 147863.8);
   zExitAccuLngthOffs : REAL := 27000.0;
   zLength_Accu_To_Z3 : REAL;
   zLength_Z1_Z2 : REAL := 148500.0;
   zStitch_Z3_To_Shear : REAL := 12600.0;
   zStitchValOffset : REAL := 15500.0;
END_VAR

ROUTINE R00_Main   (* ladder *)
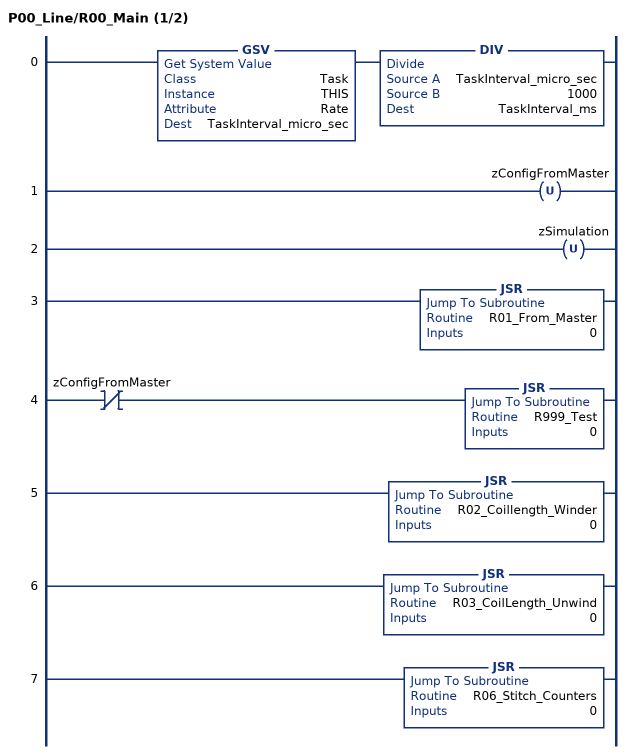
   0: GSV(Task,THIS,Rate,TaskInterval_micro_sec)DIV(TaskInterval_micro_sec,1000,TaskInterval_ms);
   1: OTU(zConfigFromMaster);
   2: OTU(zSimulation);
   3: JSR(R01_From_Master,0);
   4: XIO(zConfigFromMaster)JSR(R999_Test,0);
   5: JSR(R02_Coillength_Winder,0);
   6: JSR(R03_CoilLength_Unwind,0);
   7: JSR(R06_Stitch_Counters,0);
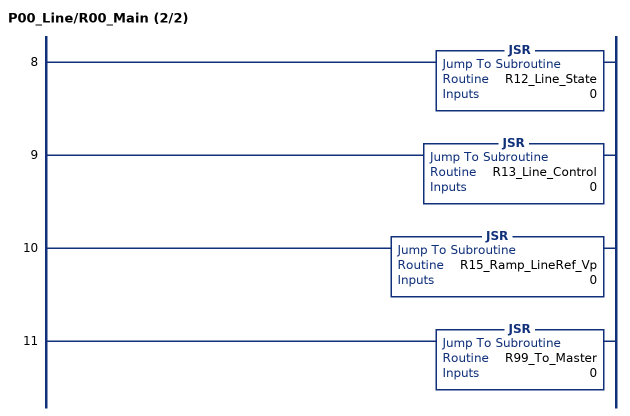
   8: JSR(R12_Line_State,0);
   9: JSR(R13_Line_Control,0);
   10: JSR(R15_Ramp_LineRef_Vp,0);
   11: JSR(R99_To_Master,0);
END_ROUTINE

ROUTINE R01_From_Master   (* ladder *)
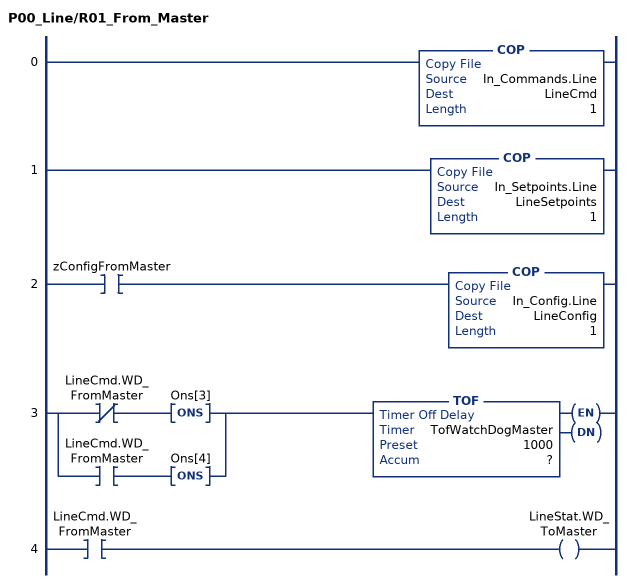
   0: COP(In_Commands.Line,LineCmd,1);
   1: COP(In_Setpoints.Line,LineSetpoints,1);
   2: XIC(zConfigFromMaster)COP(In_Config.Line,LineConfig,1);
   3: [XIO(LineCmd.WD_FromMaster) ONS(Ons[3]) ,XIC(LineCmd.WD_FromMaster) ONS(Ons[4]) ]TOF(TofWatchDogMaster,?,?);
   4: XIC(LineCmd.WD_FromMaster)OTE(LineStat.WD_ToMaster);
END_ROUTINE

ROUTINE R02_Coillength_Winder   (* ladder *)
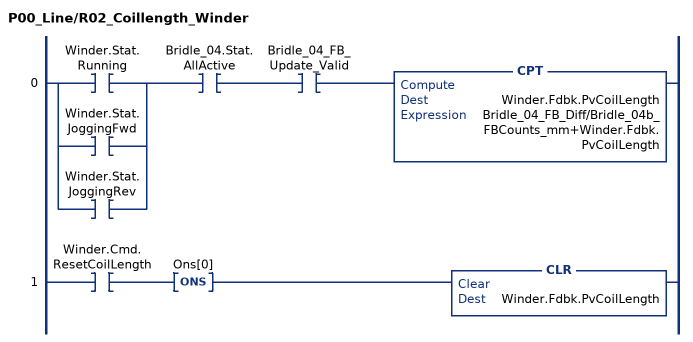
   0: [XIC(Winder.Stat.Running) ,XIC(Winder.Stat.JoggingFwd) ,XIC(Winder.Stat.JoggingRev) ]XIC(Bridle_04.Stat.AllActive)XIC(Bridle_04_FB_Update_Valid)CPT(Winder.Fdbk.PvCoilLength,Bridle_04_FB_Diff/Bridle_04b_FBCounts_mm+Winder.Fdbk.PvCoilLength);
   1: XIC(Winder.Cmd.ResetCoilLength)ONS(Ons[0])CLR(Winder.Fdbk.PvCoilLength);
END_ROUTINE

ROUTINE R03_CoilLength_Unwind   (* ladder *)
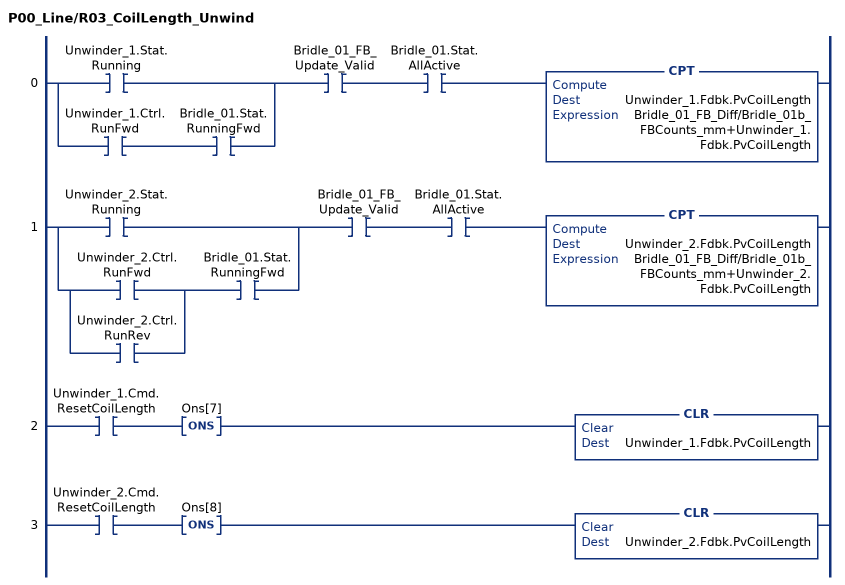
   0: [XIC(Unwinder_1.Stat.Running) ,XIC(Unwinder_1.Ctrl.RunFwd) XIC(Bridle_01.Stat.RunningFwd) ]XIC(Bridle_01_FB_Update_Valid)XIC(Bridle_01.Stat.AllActive)CPT(Unwinder_1.Fdbk.PvCoilLength,Bridle_01_FB_Diff/Bridle_01b_FBCounts_mm+Unwinder_1.Fdbk.PvCoilLength);
   1: [XIC(Unwinder_2.Stat.Running) ,[XIC(Unwinder_2.Ctrl.RunFwd) ,XIC(Unwinder_2.Ctrl.RunRev) ] XIC(Bridle_01.Stat.RunningFwd) ]XIC(Bridle_01_FB_Update_Valid)XIC(Bridle_01.Stat.AllActive)CPT(Unwinder_2.Fdbk.PvCoilLength,Bridle_01_FB_Diff/Bridle_01b_FBCounts_mm+Unwinder_2.Fdbk.PvCoilLength);
   2: XIC(Unwinder_1.Cmd.ResetCoilLength)ONS(Ons[7])CLR(Unwinder_1.Fdbk.PvCoilLength);
   3: XIC(Unwinder_2.Cmd.ResetCoilLength)ONS(Ons[8])CLR(Unwinder_2.Fdbk.PvCoilLength);
END_ROUTINE

ROUTINE R06_Stitch_Counters   (* structured text *)
   (*Initialize*)
   if s:fs then
   	Update_Cntrs_Z1:= 0;
   	Update_Cntrs_Z2:= 0;
   	ExitStat.EndAtShear:= 1;
   end_if;
   
   (*Determine arraysize*)
   Size(Stitch_Cntrs.Zone_1,0,ArrSize_Z1);
   Size(Stitch_Cntrs.Zone_2,0,ArrSize_Z2);
   
   (*Calculate mm per count*)
   Bridle_01_MM_Count:= 1/ Bridle_01b_FBCounts_mm;
   Bridle_02_MM_Count:= 1/ Bridle_02b_FBCounts_mm;
   Bridle_04_MM_Count:= 1/ Bridle_04b_FBCounts_mm;
   
   (*Validation offset*)
   StitchValPlus:= zStitchValOffset;
   StitchValMin:= - zStitchValOffset;
   
   (*Calculate material length in accumulators*)
   Entry_Accu_Mat_Length:= Entry_Accu.Fdbk.PvActualPos * 4;
   Exit_Accu_Mat_Length:= Exit_Accu.Fdbk.PvActualPos * 2;
   
   (*New stitch in line from master*)
   NewStitch_Z1_ons.InputBit:= EntryCmd.NewStitch;
   osri(NewStitch_Z1_ons);
   If NewStitch_Z1_ons.OutputBit then
   
   	If NrStitch_Z1 < ArrSize_Z1 then
   
   		NrStitch_Z1:= NrStitch_Z1 + 1;
   
   		(*Set counter to initial calculated value*)
   
   		If NrStitch_Z1 > 0 then
   			Stitch_Cntrs.Zone_1[NrStitch_Z1 - 1]:= Entry_Accu_Mat_Length + zStitcherToAccu + zEntryAccuLngthOffs;
   		end_if;
   
   	end_if;
   
   end_if;
   
   If  NrStitch_Z1 > 0 then
   
   	Indexer:= 0;
   
   	For Indexer:= 0 to NrStitch_Z1 - 1  do;
   		(*Start decrementing counter*)
   		If Bridle_02_FB_Update_Valid and Bridle_02.Stat.AllActive then
   
   			Stitch_Cntrs.Zone_1[Indexer]:= Stitch_Cntrs.Zone_1[Indexer] - (Bridle_02_FB_Diff * Bridle_02_MM_Count);
   
   		end_if;
   
   	end_for;
   
   end_if;
   
   (*Remove stitch when not detected at zone 2*)
   
   If Stitch_Cntrs.Zone_1[0] < StitchValMin then
   
   	Update_Cntrs_Z1:= 1;
   
   End_if;
   
   (*Stitch detection at Bridle 02*)
   osri(NewStitch_Z2_Ons);
   NewStitch_Z2_Ons.inputbit:= TofStitch_Z2.DN;
   
   If NewStitch_Z2_Ons.OutputBit and Bridle_02.Stat.AllActive and (Stitch_Cntrs.Zone_1[0] <> 0) then
   
   	(*Validate stitch detection*)
   
   	If (Stitch_Cntrs.Zone_1[0] > StitchValMin) and (Stitch_Cntrs.Zone_1[0] < StitchValPlus) then
   		(*If valid update table Z1*)
   		(*Increment number of stitches in Z2*)
   
   			if NrStitch_Z2 < ArrSize_Z2 then
   				NrStitch_Z2:= NrStitch_Z2 + 1;
   			end_if;
   
   		Update_Cntrs_Z1:= 1;
   
   	end_if;
   
   	(*Set max value for stitch detection at zone 3*)
   	if NrStitch_Z2 > 0 then
   		Preset_Max_Z2[NrStitch_Z2 - 1]:= Exit_Accu_Mat_Length + zLength_Z1_Z2 + zExitAccuLngthOffs;
   		(*ValCntrs_Z2[NrStitch_Z2 - 1]:= Preset_Max_Z2[NrStitch_Z2 -1];*)
   	end_if;
   end_if;
   
   Indexer:= 0;
   
   (*Count up for validation stitch detection at bridle 04*)
   
   if NrStitch_Z2 > 0 then
   	for Indexer:= 0 to NrStitch_Z2 -1 do;
   		If Bridle_04_FB_Update_Valid and Bridle_04.Stat.AllActive then
   
   			ValCntrs_Z2[Indexer]:= ValCntrs_Z2[Indexer] + (Bridle_04_FB_Diff * Bridle_04_MM_Count);
   
   		end_if;
   	end_for;
   end_if;
   
   Indexer:= 0;
   (*Update counter table for zone 1*)
   
   If Update_Cntrs_Z1 then
   
   	for Indexer:= 0 to NrStitch_Z1 do;
   
   		If Indexer < 2 then
   			Stitch_Cntrs.Zone_1[Indexer]:= Stitch_Cntrs.Zone_1[Indexer + 1];
   			Stitch_Cntrs.Zone_1[Indexer + 1]:= 0;
   		end_if;
   
   	end_for;
   
   	If NrStitch_Z1 > 0 then
   		NrStitch_Z1:= NrStitch_Z1 - 1;
   	end_if;
   
   	Update_Cntrs_Z1:= 0;
   
   end_if;
   
   Indexer:= 0;
   
   If  NrStitch_Z2 > 0 then
   
   	Indexer:= 0;
   
   	For Indexer:= 0 to NrStitch_Z2 -1  do;
   
   		If Bridle_02_FB_Update_Valid and Bridle_02.Stat.AllActive then
   
   			Stitch_Cntrs.Zone_2[Indexer]:= Stitch_Cntrs.Zone_2[Indexer] + (Bridle_02_FB_Diff * Bridle_02_MM_Count);
   
   		end_if;
   
   	end_for;
   
   end_if;
   
   (*Stitch detection at Bridle 04*)
   osri(NewStitch_Z3_Ons);
   NewStitch_Z3_Ons.inputbit:= TofStitch_Z3.dn;
   
   If NewStitch_Z3_Ons.OutputBit and Bridle_04.Stat.AllActive and (Stitch_Cntrs.Zone_2[0] <> 0) then
   
   	(*Validate stitch detection*)
   	If (ValCntrs_Z2[0] > (Preset_Max_Z2[0] + StitchValMin)) and (ValCntrs_Z2[0] < (Preset_Max_Z2[0] + StitchValPlus)) then
   		Stitch_Cntrs.Zone_3:= zStitch_Z3_To_Shear;
   		StitchIn_Z3:= 1;
   		Update_Cntrs_Z2:= 1;
   
   	end_if;
   
   
   end_if;
   
   (*Remove stitch when not detected at zone 3*)
   
   If ValCntrs_Z2[0] > (Preset_Max_Z2[0] + StitchValPlus) then
   	Update_Cntrs_Z2:= 1;
   end_if;
   
   Indexer:= 0;
   
   (*Update table with stitches from Z2*)
   
   If Update_Cntrs_Z2 then
   
   	for Indexer:= 0 to NrStitch_Z2 do;
   
   		If Indexer < 4 then
   			Stitch_Cntrs.Zone_2[Indexer]:= Stitch_Cntrs.Zone_2[Indexer + 1];
   			Stitch_Cntrs.Zone_2[Indexer + 1]:= 0;
   			Preset_Max_Z2[Indexer]:= Preset_Max_Z2[Indexer + 1];
   			Preset_Max_Z2[Indexer + 1]:= 0;
   			ValCntrs_Z2[Indexer]:= ValCntrs_Z2[Indexer + 1];
   			ValCntrs_Z2[Indexer + 1]:= 0;
   		end_if;
   
   	end_for;
   
   	If NrStitch_Z2 > 0 then
   		NrStitch_Z2:= NrStitch_Z2 - 1;
   	end_if;
   
   	Update_Cntrs_Z2:= 0;
   end_if;
   
   (*Count down to shear*)
   If Bridle_04_FB_Update_Valid and Bridle_04.Stat.AllActive and StitchIn_Z3 then
   
   	Stitch_Cntrs.Zone_3:= Stitch_Cntrs.Zone_3 - (Bridle_04_FB_Diff * Bridle_04_MM_Count);
   
   end_if;
   
   If Stitch_Cntrs.Zone_3 <  StitchValMin then
   	Stitch_Cntrs.Zone_3:= 0;
   	StitchIn_Z3:= 0;
   	ExitStat.EndAtShear:= 0;
   end_if;
   
   
   if Stitch_Cntrs.Zone_3 < 0 and StitchIn_Z3 then
   
   	ExitStat.EndAtShear:= 1;
   
   end_if;
   
   cop(Stitch_Cntrs,LineFdbks.Stitch_Cntrs,1);
END_ROUTINE
